METHOD Stop : BOOL
VAR_INPUT
END_VAR
tTimer_Enable(IN := FALSE);
tTimer_DropLid(IN := FALSE);
tTimer_Suction(IN := FALSE);
tTimer_TakeLid(IN := FALSE);
tTimer_Pick(IN := FALSE);
iCylinder_LidStopper.Extend();
iLidSuctionValve.Release();
iCupSuctionValve.Release();
END_METHOD

METHOD TakeLid : BOOL
VAR_INPUT
END_VAR
CASE nState_TakeLid OF
	0://init
		TakeLid := FALSE;
		tTimer_TakeLid(IN:= FALSE);
		tTimer_Pick(IN := FALSE);
		nState_TakeLid := 1;
	1://check LidEmpty
		IF isLidPick THEN
			IF nLine = 1 THEN
				F_SetError(51,nLine := 1);
			ELSIF nLine = 2 THEN
				F_SetError(52,nLine := 2);
			END_IF
		ELSE
			nState_TakeLid := 11;
		END_IF
	11:// call cylinder_suction. retract to take lid
		iCylinder_Suction.Retract();
		IF iCylinder_Suction.bIsRetract THEN
			tTimer_TakeLid(IN := FALSE);
			nState_TakeLid := 2;
		ELSE
			tTimer_TakeLid(IN := TRUE, PT := REAL_TO_TIME(timerCylinder_Suction)*1000);
			IF tTimer_TakeLid.Q THEN
				IF nLine = 1 THEN
					F_SetError(13,nLine := 1);
				ELSIF nLine = 2 THEN
					F_SetError(35,nLine := 2);
				END_IF
			END_IF
		END_IF
	2://call cylinder_Lidstop.retract to drop lid
		iCylinder_LidStopper.Retract();
		IF iCylinder_LidStopper.bIsRetract THEN
			tTimer_TakeLid(IN := FALSE);
			nState_TakeLid := 3;
		ELSE
			tTimer_TakeLid(IN := TRUE, PT := REAL_TO_TIME(timerCylinder_Stopper)*1000);
			IF tTimer_TakeLid.Q THEN
				IF nLine = 1 THEN
					F_SetError(11,nLine := 1);
				ELSIF nLine = 2 THEN
					F_SetError(33,nLine := 2);
				END_IF
			END_IF
		END_IF
	3:// Suck lid
		iCylinder_LidStopper.Retract();
		iLidSuctionValve.Suck();
		IF isLidPick THEN
			tTimer_TakeLid(IN := FALSE);
			nState_TakeLid := 33;
		ELSE
			tTimer_TakeLid(IN := TRUE, PT := REAL_TO_TIME(timerCheckLidSuck)*1000);
			IF tTimer_TakeLid.Q THEN
				IF nLine = 1 THEN
					F_SetError(49,nLine := 1);
					nState_TakeLid := 2;
				ELSIF nLine = 2 THEN
					F_SetError(50,nLine := 2);
					nState_TakeLid := 2;
				END_IF
			END_IF
		END_IF
	33:
		iLidSuctionValve.Suck();
		tTimer_Pick(IN := TRUE, PT:= T#0.5S);
		IF tTimer_Pick.Q THEN
			nState_TakeLid := 4;
		END_IF
	4://Block Lid Up
		iLidSuctionValve.Suck();
		tTimer_Pick(IN := FALSE);
		iCylinder_LidStopper.Extend();
		IF iCylinder_LidStopper.bIsExtend THEN
			tTimer_TakeLid(IN := FALSE);
			nState_TakeLid := 5;
		ELSE
			tTimer_TakeLid(IN := TRUE, PT := REAL_TO_TIME(timerCylinder_Stopper)*1000);
			IF tTimer_TakeLid.Q THEN
				IF nLine = 1 THEN
					F_SetError(12,nLine := 1);
				ELSIF nLine = 2 THEN
					F_SetError(34,nLine := 2);
				END_IF
			END_IF
		END_IF
	5://finish takelid
		TakeLid := TRUE;
		nState_TakeLid := 0;	
END_CASE
END_METHOD

END_FUNCTION_BLOCK

// ---- POUs/Components/Child Components/FB_SuctionCup.TcPOU
FUNCTION_BLOCK FB_SuctionCup IMPLEMENTS I_SuctionCup
VAR_INPUT
END_VAR
VAR_OUTPUT
END_VAR
VAR
	fPressure 		AT %I*	: REAL;
	bSuck			AT %Q*	: BOOL;
	bPressure		AT %I* 	: BOOL;
END_VAR

PROPERTY bIsSuck : BOOL
GET
bIsSuck := bPressure;
END_GET
END_PROPERTY

PROPERTY fThreshold : REAL
GET
fThreshold := 6;
END_GET
SET
END_SET
END_PROPERTY

METHOD Release : BOOL
VAR_INPUT
END_VAR
bSuck := FALSE;
END_METHOD

METHOD Suck : BOOL
VAR_INPUT
END_VAR
bSuck := TRUE;
END_METHOD

END_FUNCTION_BLOCK

// ---- POUs/Components/Sim Components/FB_SuctionCup_Sim.TcPOU
FUNCTION_BLOCK FB_SuctionCup_Sim IMPLEMENTS I_SuctionCup
VAR_INPUT
END_VAR
VAR_OUTPUT
END_VAR
VAR
	fPressure 			: REAL;// Value 0-100 %
	bSuck				: BOOL;
	// var sim
	tTimer				: TON;
	tDelay				: TIME := T#1000MS;// acceleration time of fPressure to value = 100
	nState				: INT := 0;
	bRelease			: BOOL := TRUE;
END_VAR

CASE nState OF
	0: //init release Suction
		IF bRelease THEN
			bSuck := FALSE;
			fPressure := 0;
		ELSE
			bSuck := TRUE;
			fPressure := 100;
		END_IF
		tTimer(IN := FALSE);
		nState := nState + 1;
	1:// check for signal
		tTimer(IN := FALSE);
		IF bSuck AND (fPressure = 0) THEN
			nState := 10;
		END_IF
		IF NOT bSuck AND (fPressure = 100) THEN
			nState := 20;
		END_IF
	10: //Suck 
		tTimer(IN := TRUE,PT := tDelay);
		fPressure := TIME_TO_REAL(tTimer.ET)*(100/TIME_TO_REAL(tDelay));
		IF (fPressure = 100) THEN
			nState := 1;
		END_IF
	20:// release
		tTimer(IN := TRUE,PT := tDelay);
		fPressure := 100 - (TIME_TO_REAL(tTimer.ET)*(100/TIME_TO_REAL(tDelay)));
		IF (fPressure = 0) THEN
			nState := 1;
		END_IF
END_CASE

PROPERTY bIsSuck : BOOL
GET
IF fPressure > fThreshold THEN
	bIsSuck := TRUE;
ELSE 
	bIsSuck := FALSE;
END_IF
END_GET
END_PROPERTY

PROPERTY fThreshold : REAL
GET
fThreshold := 50;
END_GET
SET
END_SET
END_PROPERTY

METHOD Release : BOOL
VAR_INPUT
END_VAR
bSuck := FALSE;
END_METHOD

METHOD Suck : BOOL
VAR_INPUT
END_VAR
bSuck := TRUE;
END_METHOD

END_FUNCTION_BLOCK

// ---- POUs/Modules/FB_LidCloseModule.TcPOU
FUNCTION_BLOCK FB_LidCloseModule
VAR_INPUT
	nLine							: INT;
	timer_Check_Cylinder_extend		: REAL;
	timer_Check_Cylinder_retract	: REAL;
	timer_CloseLid					: REAL;
END_VAR
VAR_OUTPUT
END_VAR
VAR
	// ===== CHILD COMPONENTS ======
	fbCylinder_LidClose 		: FB_Cylinder;
	// ===== SIM COMPONENTS ======
	fbCylinder_LidClose_Sim		: FB_Cylinder_Sim;
	// ===== INTERFACES ======
	iCylinder					: I_Cylinder;
	// ===== Var method enable
	nState_Enable				: INT;
	tTimer_Enable				: TON;
	// ===== Var method CloseLid
	nState_Close				: INT;
	tTimer_Close				: TON;
	i							: INT := 1; //number of repetitions
END_VAR

IF bSimMode THEN
	iCylinder := fbCylinder_LidClose_Sim;
	fbCylinder_LidClose_Sim();
ELSE
	iCylinder := fbCylinder_LidClose;
	fbCylinder_LidClose(id := 1);
END_IF

METHOD CloseLid : BOOL
VAR_INPUT
END_VAR
CASE nState_Close OF
	0:
		CloseLid := FALSE;
		tTimer_Close(IN := FALSE);
		nState_Close := 1;
	1: //set init i
		i := 1;
		nState_Close := 2;
	2: // cylinder extend and check sensor
		iCylinder.Extend();
		IF iCylinder.bIsExtend THEN
			tTimer_Close(IN := FALSE);
			nState_Close := 3;
		ELSE
			tTimer_Close(IN := TRUE,PT := REAL_TO_TIME(timer_Check_Cylinder_extend)*1000);
			IF tTimer_Close.Q THEN
				i := i + 1;
				nState_Close := 3;
			END_IF
		END_IF
	3: //cylinder retract
		iCylinder.Retract();
		IF iCylinder.bIsRetract THEN
			tTimer_Close(IN := FALSE);
			nState_Close := 4;//return extend
		ELSE
			tTimer_Close(IN := TRUE,PT := REAL_TO_TIME(timer_Check_Cylinder_retract)*1000);
			IF tTimer_Close.Q THEN
				IF nLine = 1 THEN
					F_SetError(15,nLine := 1);
				ELSIF nLine = 2 THEN
					F_SetError(37,nLine := 2);
				END_IF
			END_IF
		END_IF
	4:// cylinder extend and check sensor
		iCylinder.Extend();
		IF iCylinder.bIsExtend THEN
			tTimer_Close(IN := FALSE);
			nState_Close := 5;
		ELSE
			tTimer_Close(IN := TRUE,PT := REAL_TO_TIME(timer_Check_Cylinder_extend)*1000);
			IF tTimer_Close.Q THEN
				i := i + 1;
				nState_Close := 5;
			END_IF
		END_IF
	5:// cylinder retract -> end
		iCylinder.Retract();
		IF iCylinder.bIsRetract THEN
			tTimer_Close(IN := FALSE);
			nState_Close := 6;//end
		ELSE
			tTimer_Close(IN := TRUE,PT := REAL_TO_TIME(timer_Check_Cylinder_retract)*1000);
			IF tTimer_Close.Q THEN
				IF nLine = 1 THEN
					F_SetError(15,nLine := 1);
				ELSIF nLine = 2 THEN
					F_SetError(37,nLine := 2);
				END_IF
			END_IF
		END_IF
	6://check warning
		IF (i = 3) THEN
			IF nLine = 1 THEN
				F_SetWarning(107,nLine := 1);
			ELSIF nLine = 2 THEN 
				F_SetWarning(114,nLine := 2);
			END_IF
			
			nState_Close := 7; //end
		ELSE
			nState_Close := 7; //end
		END_IF
	7: //Finish
		CloseLid := TRUE;
		nState_Close := 0;
END_CASE
END_METHOD

METHOD Enable : BOOL
VAR_INPUT
END_VAR
CASE nState_Enable OF
	0:
		Enable 			:= FALSE;
		tTimer_Enable(IN := FALSE);
		nState_Enable 	:= 1;
	1: // cylinder retract and check
		iCylinder.Retract();
		IF iCylinder.bIsRetract THEN
			tTimer_Enable(IN := FALSE);
			nState_Enable 	:= 2;
		ELSE
			tTimer_Enable(IN := TRUE, PT := REAL_TO_TIME(timer_Check_Cylinder_retract)*1000);
			IF tTimer_Enable.Q THEN
				IF nLine = 1 THEN
					F_SetError(15,nLine := 1);
				ELSIF nLine = 2 THEN
					F_SetError(33,nLine := 2);
				END_IF
			END_IF
		END_IF
	2:
		tTimer_Enable(IN := FALSE);
		Enable := TRUE;
	99://Error
END_CASE
END_METHOD

METHOD Init : BOOL
VAR_INPUT
END_VAR
nState_Close := 0;
i 			 := 1;
END_METHOD

METHOD Manual : BOOL
VAR_INPUT
	bCylinder_CloseLid_Extend	: BOOL;
	bCylinder_CloseLid_Retract	: BOOL;
END_VAR
IF bCylinder_CloseLid_Extend THEN
	iCylinder.Extend();
	IF iCylinder.bIsExtend THEN
		tTimer_Close(IN := FALSE);
	ELSE
		tTimer_Close(IN := TRUE,PT := REAL_TO_TIME(timer_Check_Cylinder_retract)*1000);
		IF tTimer_Close.Q THEN
			IF nLine = 1 THEN
				F_SetError(16,nLine := 1);
			ELSIF nLine = 2 THEN
				F_SetError(38,nLine := 2);
			END_IF
		END_IF
	END_IF
ELSIF bCylinder_CloseLid_Retract THEN
	iCylinder.Retract();
	IF iCylinder.bIsRetract THEN
		tTimer_Close(IN := FALSE);
	ELSE
		tTimer_Close(IN := TRUE,PT := REAL_TO_TIME(timer_Check_Cylinder_retract)*1000);
		IF tTimer_Close.Q THEN
			IF nLine = 1 THEN
				F_SetError(15,nLine := 1);
			ELSIF nLine = 2 THEN
				F_SetError(37,nLine := 2);
			END_IF
		END_IF
	END_IF
END_IF
END_METHOD

METHOD Reset : BOOL
VAR_INPUT
END_VAR
tTimer_Enable(IN := FALSE);							
tTimer_Close(IN := FALSE);
iCylinder.Retract();
END_METHOD

METHOD Stop : BOOL
VAR_INPUT
END_VAR
tTimer_Enable(IN := FALSE);						
tTimer_Close(IN := FALSE);
END_METHOD

END_FUNCTION_BLOCK

// ---- POUs/Modules/FB_Transfer.TcPOU
FUNCTION_BLOCK FB_Transfer
VAR_INPUT
	nLine					: INT;
	fTimer_Comb				: REAL;
	fTimer_Clip				: REAL;
	fTimer_Move_Comb		: REAL;
END_VAR
VAR_OUTPUT
	nDoneTransfer			: INT;
	bDoneTransfer			: BOOL;
END_VAR
VAR
	fbCylinder_Comb			: FB_Cylinder;
	fbCylinder_Clip			: FB_Cylinder;
	fbCylinder_Move_Comb	: FB_Cylinder;
	// ===== SIM COMPONENTS ==============
	fbCylinderSim_Comb		: FB_Cylinder_Sim;
	fbCylinderSim_Clip		: FB_Cylinder_Sim;
	fbCylinderSim_Move_Comb	: FB_Cylinder_Sim;
	// ===== INTERFACES ==================
	iCylinder_Comb			: I_Cylinder;
	iCylinder_Clip			: I_Cylinder;
	iCylinder_Move_Comb		: I_Cylinder;
	//====== VAR MOTHOD ==================
	nState					: INT;
	nStateEnable			: INT;
	nState_Reset			: INT;
	tTimer_Reset			: TON;
	fbTimer_Comb			: TON;
	fbTimer_Clip			: TON;
	fbTimer_Move_Comb		: TON;
	//======== VAR HMI Transfer Setting ====
END_VAR

IF bSimMode THEN
	iCylinder_Clip 	:= fbCylinderSim_Clip;
	fbCylinderSim_Clip();
	iCylinder_Comb	:= fbCylinderSim_Comb;
	fbCylinderSim_Comb();
	iCylinder_Move_Comb	:= fbCylinderSim_Move_Comb;
	fbCylinderSim_Move_Comb();
ELSE
	iCylinder_Clip 	:= fbCylinder_Clip;
	fbCylinder_Clip(id := 1);
	iCylinder_Comb	:= fbCylinder_Comb;
	fbCylinder_Comb(id := 1);
	iCylinder_Move_Comb	:= fbCylinder_Move_Comb;
	fbCylinder_Move_Comb(id := 1);
END_IF

METHOD Auto : BOOL
VAR_INPUT
END_VAR
fbTimer_Clip(PT := REAL_TO_TIME(fTimer_Clip)*1000);
fbTimer_Comb(PT := REAL_TO_TIME(fTimer_Comb)*1000);
fbTimer_Move_Comb(PT := REAL_TO_TIME(fTimer_Move_Comb)*1000);
CASE nState OF 
	0: // init value
		Auto		:= FALSE;
		fbTimer_Move_Comb(IN := FALSE);
		fbTimer_Clip(IN	:= FALSE);
		fbTimer_Comb(IN	:= FALSE);
		nState		:= 1;
	1: // Cylinder Clip and Comb Extend hold cup
		bDoneTransfer 	:= FALSE;
		iCylinder_Clip.Extend();
		iCylinder_Comb.Extend();
		fbTimer_Clip(IN	:= TRUE);
		fbTimer_Comb(IN	:= TRUE);
		IF iCylinder_Clip.bIsExtend AND iCylinder_Comb.bIsExtend THEN
			nState	:= 2;
		ELSIF fbTimer_Comb.Q AND NOT fbTimer_Clip.Q THEN
			IF nLine = 1 THEN
				F_SetError(18,nLine := 1);
			ELSIF nLine = 2 THEN
				F_SetError(40,nLine := 2);
			END_IF
		ELSIF fbTimer_Clip.Q AND NOT fbTimer_Comb.Q THEN
			IF nLine = 1 THEN
				F_SetError(20,nLine := 1);
			ELSIF nLine = 2 THEN
				F_SetError(42,nLine := 2);
			END_IF
		ELSIF iCylinder_Clip.bIsExtend AND fbTimer_Comb.Q THEN
			IF nLine = 1 THEN
				F_SetError(18,nLine := 1);
			ELSIF nLine = 2 THEN
				F_SetError(40,nLine := 2);
			END_IF
		ELSIF iCylinder_Comb.bIsExtend AND fbTimer_Clip.Q THEN
			IF nLine = 1 THEN
				F_SetError(20,nLine := 1);
			ELSIF nLine = 2 THEN
				F_SetError(42,nLine := 2);
			END_IF
		ELSIF fbTimer_Comb.Q AND fbTimer_Clip.Q THEN
			IF nLine = 1 THEN
				F_SetError(18,nLine := 1);
			ELSIF nLine = 2 THEN
				F_SetError(40,nLine := 2);
			END_IF
		END_IF
	2: // Cylinder_Move_Comb Extend move cup
		fbTimer_Clip(IN	:= FALSE);
		fbTimer_Comb(IN	:= FALSE);
		fbTimer_Move_Comb(IN := TRUE);
		iCylinder_Move_Comb.Extend();
		IF iCylinder_Move_Comb.bIsExtend THEN
			nState	:= 3;
		ELSIF fbTimer_Move_Comb.Q THEN
			IF nLine = 1 THEN
				F_SetError(22,nLine := 1);
			ELSIF nLine = 2 THEN
				F_SetError(44,nLine := 2);
			END_IF
		END_IF
	3: // retract clip and comb
		fbTimer_Comb(IN := TRUE);
		fbTimer_Move_Comb(IN := FALSE);
		iCylinder_Comb.Retract();
		IF iCylinder_Comb.bIsRetract THEN
			nState	:= 33;
		ELSIF fbTimer_Comb.Q THEN
			IF nLine = 1 THEN
				F_SetError(17,nLine := 1);
			ELSIF nLine = 2 THEN
				F_SetError(39,nLine := 2);
			END_IF
		END_IF
	33:
		fbTimer_Clip(IN := TRUE);
		fbTimer_Comb(IN := FALSE);
		iCylinder_Clip.Retract();
		IF iCylinder_Clip.bIsRetract THEN
			nDoneTransfer	:= nDoneTransfer + 1;
			bDoneTransfer 	:= TRUE;
			IF nLine = 1 THEN 
				bToDropcup1			:= TRUE;
			ELSIF nLine = 2 THEN
				bToDropcup2			:= TRUE;
			END_IF
			IF nDoneTransfer > 8 THEN
				nDoneTransfer := 8;
			END_IF
			nState	:= 4;
		ELSIF fbTimer_Clip.Q THEN
			IF nLine = 1 THEN
				F_SetError(19,nLine := 1);
			ELSIF nLine = 2 THEN
				F_SetError(41,nLine := 2);
			END_IF
		END_IF
	4://Move_Comb Retract
		fbTimer_Clip(IN := FALSE);
		fbTimer_Move_Comb(IN := TRUE);
		iCylinder_Move_Comb.Retract();
		IF iCylinder_Move_Comb.bIsRetract THEN
			nState	:= 5;
		ELSIF fbTimer_Move_Comb.Q THEN
			IF nLine = 1 THEN
				F_SetError(21,nLine := 1);
			ELSIF nLine = 2 THEN
				F_SetError(43,nLine := 2);
			END_IF
		END_IF
	5:// Complete
		fbTimer_Move_Comb(IN := FALSE);
		Auto		:= TRUE;
		nState		:= 0;	
END_CASE
END_METHOD

METHOD Enable : BOOL
VAR_INPUT
END_VAR
fbTimer_Clip(PT := REAL_TO_TIME(fTimer_Clip)*1000);
fbTimer_Comb(PT := REAL_TO_TIME(fTimer_Comb)*1000);
fbTimer_Move_Comb(PT := REAL_TO_TIME(fTimer_Move_Comb)*1000);
CASE nStateEnable OF
	0:// init 
		Enable					:= FALSE;
		fbTimer_Clip(IN	:= FALSE);
		fbTimer_Comb(IN	:= FALSE);
		fbTimer_Move_Comb(IN := FALSE);
		nStateEnable			:= 1;
	1:// Retract Comb and Clip
		iCylinder_Clip.Retract();
		iCylinder_Comb.Retract();
		fbTimer_Clip(IN	:= TRUE);
		fbTimer_Comb(IN	:= TRUE);
		IF iCylinder_Clip.bIsRetract AND iCylinder_Comb.bIsRetract THEN
			nStateEnable		:= 2;
		ELSIF fbTimer_Clip.Q AND NOT fbTimer_Comb.Q THEN
			nStateEnable		:= 10;
		ELSIF fbTimer_Comb.Q AND NOT fbTimer_Clip.Q THEN
			nStateEnable		:= 11;
		END_IF	
	2:// Retract MoveComb
		fbTimer_Clip(IN	:= FALSE);
		fbTimer_Comb(IN	:= FALSE);
		iCylinder_Move_Comb.Retract();
		fbTimer_Move_Comb.IN	:= TRUE;
		IF iCylinder_Move_Comb.bIsRetract THEN
			nStateEnable		:= 3;
		ELSIF fbTimer_Move_Comb.Q THEN
			nState				:= 12;
		END_IF
	3:// Enable
		fbTimer_Move_Comb(IN := FALSE);
		Enable					:= TRUE;
	10:// Error Cylinder Clip
		IF nLine = 1 THEN
			F_SetError(17,nLine := 1);
			nState	:= 99;
		ELSIF nLine = 2 THEN
			F_SetError(35,nLine := 2);
			nState	:= 99;
		END_IF
	11:// Error Cylinder Comb
		IF nLine = 1 THEN
			F_SetError(16,nLine := 1);
			nState	:= 99;
		ELSIF nLine = 2 THEN
			F_SetError(34,nLine := 2);
			nState	:= 99;
		END_IF
	12:// Error Cylinder MoveComb
		IF nLine = 1 THEN
			F_SetError(18,nLine := 1);
			nState	:= 99;
		ELSIF nLine = 2 THEN
			F_SetError(36,nLine := 2);
			nState	:= 99;
		END_IF
	99:// Error
END_CASE
END_METHOD

METHOD Init : BOOL
VAR_INPUT
END_VAR
nState		 := 0;
nStateEnable := 0;
bDoneTransfer := FALSE;
nDoneTransfer := 0;
END_METHOD

METHOD Manual : BOOL
VAR_INPUT
	bCylinder_Comb_Extend			: BOOL;
	bCylinder_Comb_Retract			: BOOL;
	bCylinder_Clip_Extend			: BOOL;
	bCylinder_Clip_Retract			: BOOL;
	bCylinder_Move_Comb_Extend		: BOOL;
	bCylinder_Move_Comb_Retract		: BOOL;
END_VAR
IF bCylinder_Comb_Extend THEN
	iCylinder_Comb.Extend();
	IF iCylinder_Comb.bIsExtend THEN
		fbTimer_Comb(IN := FALSE);
	ELSE
		fbTimer_Comb(PT := REAL_TO_TIME(fTimer_Comb)*1000);
			IF fbTimer_Comb.Q THEN
				IF nLine = 1 THEN
					F_SetError(18,nLine := 1);
				ELSIF nLine = 2 THEN
					F_SetError(40,nLine := 2);
				END_IF
			END_IF
	END_IF
END_IF

IF bCylinder_Comb_Retract THEN
	iCylinder_Comb.Retract();
	IF iCylinder_Comb.bIsRetract THEN
		fbTimer_Comb(IN := FALSE);
	ELSE
		fbTimer_Comb(PT := REAL_TO_TIME(fTimer_Comb)*1000);
			IF fbTimer_Comb.Q THEN
				IF nLine = 1 THEN
					F_SetError(17,nLine := 1);
				ELSIF nLine = 2 THEN
					F_SetError(39,nLine := 2);
				END_IF
			END_IF
	END_IF
END_IF

IF bCylinder_Clip_Extend THEN
	iCylinder_Clip.Extend();
	IF iCylinder_Clip.bIsExtend THEN
		fbTimer_Clip(IN := FALSE);
	ELSE
		fbTimer_Clip(PT := REAL_TO_TIME(fTimer_Clip)*1000);
			IF fbTimer_Clip.Q THEN
				IF nLine = 1 THEN
					F_SetError(20,nLine := 1);
				ELSIF nLine = 2 THEN
					F_SetError(42,nLine := 2);
				END_IF
			END_IF
	END_IF
END_IF


IF bCylinder_Clip_Retract THEN
	iCylinder_Clip.Retract();	
	IF iCylinder_Clip.bIsRetract THEN
		fbTimer_Clip(IN := FALSE);
	ELSE
		fbTimer_Clip(PT := REAL_TO_TIME(fTimer_Clip)*1000);
			IF fbTimer_Clip.Q THEN
				IF nLine = 1 THEN
					F_SetError(19,nLine := 1);
				ELSIF nLine = 2 THEN
					F_SetError(41,nLine := 2);
				END_IF
			END_IF
	END_IF
END_IF

IF bCylinder_Move_Comb_Extend THEN
	iCylinder_Move_Comb.Extend();
	IF iCylinder_Move_Comb.bIsExtend THEN
		fbTimer_Move_Comb(IN := FALSE);
	ELSE
		fbTimer_Move_Comb(PT := REAL_TO_TIME(fTimer_Move_Comb)*1000);
			IF fbTimer_Move_Comb.Q THEN
				IF nLine = 1 THEN
					F_SetError(22,nLine := 1);
				ELSIF nLine = 2 THEN
					F_SetError(44,nLine := 2);
				END_IF
			END_IF
	END_IF
END_IF

IF bCylinder_Move_Comb_Retract THEN
	iCylinder_Move_Comb.Retract();
	IF iCylinder_Move_Comb.bIsRetract THEN
		fbTimer_Move_Comb(IN := FALSE);
	ELSE
		fbTimer_Move_Comb(PT := REAL_TO_TIME(fTimer_Move_Comb)*1000);
			IF fbTimer_Move_Comb.Q THEN
				IF nLine = 1 THEN
					F_SetError(21,nLine := 1);
				ELSIF nLine = 2 THEN
					F_SetError(43,nLine := 2);
				END_IF
			END_IF
	END_IF
END_IF
END_METHOD

METHOD Reset : BOOL
VAR_INPUT
END_VAR
iCylinder_Clip.Retract();
fbTimer_Clip(IN	:= FALSE);
fbTimer_Comb(IN	:= FALSE);
fbTimer_Move_Comb(IN := FALSE);

CASE nState_Reset OF
	0:
		iCylinder_Comb.Retract();
		tTimer_Reset(IN := TRUE, PT := T#300MS);
		IF tTimer_Reset.Q OR iCylinder_Comb.bIsRetract THEN
			nState_Reset := 1;
		END_IF
	1:
		iCylinder_Move_Comb.Retract();
		nState_Reset := 0;
END_CASE
END_METHOD

METHOD Stop : BOOL
VAR_INPUT
END_VAR
fbTimer_Clip(IN	:= FALSE);
fbTimer_Comb(IN	:= FALSE);
fbTimer_Move_Comb(IN := FALSE);
END_METHOD

END_FUNCTION_BLOCK

// ---- POUs/Machines/PR_Line02.TcPOU
PROGRAM PR_Line02
VAR PERSISTENT
//----------------VAR SETTING--------------------
	timerCheckCylinder_Up			: REAL;//CupSupply
	timerCheckCylinder_Dw			: REAL;
	timerCheckEmpty					: REAL;
	timerCheckStuck					: REAL;
	timerCylinder_Up_extend 		: REAL;
	timerCylinder_Suction_Cup_extend: REAL;
	timerCylinder_Suction_Cup		: REAL;
	timerCylinder_Suction_Val		: REAL;
	timerCylinder_Suction_pick		: REAL;
	fSpeed_motor_mixer				: REAL;//FoodMixer
	fTimer_Reverse					: REAL;
	fFast_Speed						: REAL;//FoodWeight
	fSlow_Speed_1					: REAL;
	fSlow_Speed_2					: REAL;
	fDerisedWeight_Food				: REAL;
	fChangeMode_Food_1				: REAL;
	fChangeMode_Food_2				: REAL;
	fMaxWeight_Food					: REAL;
	fPerStop_Food					: REAL;
	fTimer_Food						: REAL;
	fTimer_Alarm_Food				: REAL;
	fTimer_Check_Food				: REAL;
	fDelta_Food						: REAL;
	fTimer_rever_food				: REAL;
	fTimer_Error_Food				: REAL;
	fFast_Speed_vibrating_funnel	: REAL;//WormWeight
	fSlow_Speed_vibrating_funnel_1	: REAL;
	fSlow_Speed_vibrating_funnel_2	: REAL;
	fDerisedWeight_Worm				: REAL;
	fChangeMode_Worm_1				: REAL;
	fChangeMode_Worm_2				: REAL;
	fMaxWeight_Worm					: REAL;
	fPerStop_Worm					: REAL;
	fTimer_Worm						: REAL;
	fTimer_Alarm_Worm				: REAL;
	fTimer_Check_Worm				: REAL;
	fTimer_Check_Cylinder			: REAL;
	fDelta_Worm						: REAL;
	fTimer_Error_Worm				: REAL;
	timerCylinder_Suction			: REAL;//LidSupply
	timerCheckLidRelease			: REAL;
	timerLidBlow					: REAL;
	timerCheckLidEmpty				: REAL;
	timerCheckLidSuck				: REAL;
	timerCylinder_Stopper			: REAL;
	timer_Check_Cylinder_extend		: REAL;//LidClose
	timer_Check_Cylinder_retract	: REAL;
	timer_CloseLid					: REAL;
	fTimer_Comb						: REAL;//Transfer
	fTimer_Clip						: REAL;
	fTimer_Move_Comb				: REAL;
//-----------------VAR HMI-------------------
	fProductLog						: ARRAY [1..2] OF ARRAY  [1..5] OF REAL;
END_VAR

VAR
	bStatus_Food					: BOOL;
	bStatus_Worm					: BOOL;
//----------------VAR MANUAL---------------------
	bCylinder_up_extend 			: BOOL;//CupSupply
	bCylinder_up_retract 			: BOOL;
	bCylinder_dw_extend 			: BOOL;
	bCylinder_dw_retract 			: BOOL;
	bCylinder_Suction_cup_extend	: BOOL;
	bCylinder_Suction_cup_retract	: BOOL;
	bUp_Motor_Mixer					: BOOL;//FoodMixer
	bDown_Motor_Mixer				: BOOL;
	bMotor_mixer_Manual				: BOOL;
	bMotor_mixer_reverse			: BOOL;
	bUp_Food_Motor					: BOOL;//FoodWeight
	bDown_Food_Motor				: BOOL;
	bZero_Loadcell_Food				: BOOL;
	bMotor_Food						: BOOL;
	bMotor_Food_reverse				: BOOL;
	bUp_vibrating_funnel			: BOOL;//WormWeight
	bDown_vibrating_funnel			: BOOL;
	bZero_Loadcell_Worm				: BOOL;
	bCylinder_Block_Worm_Extend		: BOOL;
	bCylinder_Block_Worm_Retract	: BOOL;
	bMotor_vibrating_funnel			: BOOL;	
	bCylinder_LidStopper_extend 	: BOOL;//LidSupply
	bCylinder_LidStopper_retract 	: BOOL;
	bCylinder_Suction_extend		: BOOL;
	bCylinder_Suction_retract		: BOOL;
	bLidSuctionValve				: BOOL;
	bCupSuctionValve				: BOOL;
	bBlowValve						: BOOL;
	bCylinder_CloseLid_Extend		: BOOL;//LidClose
	bCylinder_CloseLid_Retract		: BOOL;
	bCylinder_Comb_Extend			: BOOL;//Transfer
	bCylinder_Comb_Retract			: BOOL;
	bCylinder_Clip_Extend			: BOOL;
	bCylinder_Clip_Retract			: BOOL;
	bCylinder_Move_Comb_Extend		: BOOL;
	bCylinder_Move_Comb_Retract		: BOOL;
//------------------fbmodule----------------
	fb_CupSupply	: FB_CupSupplyModule;
	fb_FoodMixer	: FB_FoodMixerModule;
	fb_FoodWeight	: FB_FoodWeightModule;
	fb_WormWeight	: FB_WormWeightModule;
	fb_LidSupply	: FB_LidSupplyModule;
	fb_LidClose		: FB_LidCloseModule;
	fb_Transfer		: FB_Transfer;
//---------------- VAR Method ---------------
	nState				: INT;
	nState_Dropcup		: INT;
	nState_Transfer		: INT;
	nState_FoodWeight	: INT;
	nState_WormWeight	: INT;
	nState_LidClose		: INT;
	nState_LidSupply	: INT;
	nDoneTransfer		: INT;
	nDoneTransferStop	: INT;
	tmp					: INT;
	bDoneTakeLid		: BOOL;
	bDoneTransfer		: BOOL;
	bDoneCupSupply		: BOOL;
	bDoneFoodWeight		: BOOL;
	bDoneWormWeight		: BOOL;
	bDoneLidSupply		: BOOL;
	bDoneLidClose		: BOOL;
	bEnable				: BOOL;
	bFinishCupSupply	: BOOL;
	bFinishFoodWeight	: BOOL;
	bFinishWormWeight	: BOOL;
	bFinishLidSupply	: BOOL;
	bFinishLidClose		: BOOL;
	bFinishTransfer		: BOOL;
	//-------VAR--------------
	nStateConveyor		: INT;
	fbtimertransfer		: TON;
	fbTimer				: TON;
	nStateStop			: INT;
	fbtimerStop			: ton;
	fbTimerCycle		: ton;
	timeCycle			: REAL :=1;
	fproduct			: INT;
	nstateCycle			: INT;
	bDone				: R_TRIG;
	fbDelay				: TON;
	bStatus_Food_order	: ARRAY [1..3] OF BOOL;
	bStatus_Worm_order	: ARRAY [1..3] OF BOOL;
	bStatus_Lid_order	: ARRAY [1..3] OF BOOL;
	i1,i2,i3			: INT := 0;
	xathucan			: BOOL;
	xasau				: BOOL;
	daothucan			: BOOL;
	nstatetest1			: INT;
	nstatetest2			: INT;
	nstatetest3			: INT;
	bxa					: BOOL;
	bCheck				: BOOL;
	bypassFood			: BOOL;
	bypassWorm			: BOOL;
	bypassLid			: BOOL;
END_VAR

fb_CupSupply(
	nLine:= 2 , 
	timerCheckCylinder_Up:= timerCheckCylinder_Up, 
	timerCheckCylinder_Dw:= timerCheckCylinder_Dw, 
	timerCheckEmpty:= timerCheckEmpty, 
	timerCheckStuck:= timerCheckStuck,
	timerCylinder_Up_extend := timerCylinder_Up_extend,
	timerCylinder_Suction:= timerCylinder_Suction_Cup,
	timerCylinder_Suction_extend:= timerCylinder_Suction_Cup_extend,
	ttimerCylinder_val:=timerCylinder_Suction_Val,
	timerCylinder_Suction_pick:=timerCylinder_Suction_pick);

fb_FoodMixer(
	nLine:= 2,
	UnitID:= 1, 
	fSpeed_motor_mixer:= fSpeed_motor_mixer,
	fTimer_Reverse:= fTimer_Reverse);
		
fb_FoodWeight(
	nLine:= 2, 
	UnitID:= 6, 
	fFast_Speed:= fFast_Speed, 
	fSlow_Speed_1:= fSlow_Speed_1, 
	fSlow_Speed_2:= fSlow_Speed_2, 
	fDerisedWeight_Food:= fDerisedWeight_Food, 
	fChangeMode_Food_1:= fChangeMode_Food_1, 
	fChangeMode_Food_2:= fChangeMode_Food_2, 
	fMaxWeight_Food:= fMaxWeight_Food, 
	fPerStop_Food:= fPerStop_Food, 
	fTimer_Food:= fTimer_Food, 
	fTimer_Alarm_Food:= fTimer_Alarm_Food, 
	fTimer_Check_Food:= fTimer_Check_Food, 
	fDelta_Food:= fDelta_Food,
	fTimer_Reverse := fTimer_rever_food,
	fTimer_Error_Food := fTimer_Error_Food, 
	fProductLogF=> fProductLog[1],
	bStatus_Food=> bStatus_Food,
	Time_start=>Time_Start_Food_line2,
	Time_Stop=>Time_Stop_Food_line2,
	status=>bStatus_Food_line2,
	fweight_iot =>fWeight_Food_line2);

fb_LidClose(
	nLine:= 2, 
	timer_Check_Cylinder_extend:= timer_Check_Cylinder_extend, 
	timer_Check_Cylinder_retract:= timer_Check_Cylinder_retract, 
	timer_CloseLid:= timer_CloseLid);
	
fb_LidSupply(
	nLine:= 2, 
	timerCylinder_Suction:= timerCylinder_Suction, 
	timerCheckLidRelease:= timerCheckLidRelease, 
	timerLidBlow:= timerLidBlow, 
	timerCheckLidEmpty:= timerCheckLidEmpty, 
	timerCheckLidSuck:= timerCheckLidSuck, 
	timerCylinder_Stopper:= timerCylinder_Stopper);

fb_Transfer(
	nLine:= 2, 
	fTimer_Comb:= fTimer_Comb, 
	fTimer_Clip:= fTimer_Clip, 
	fTimer_Move_Comb:= fTimer_Move_Comb, 
	nDoneTransfer=> nDoneTransfer,
	bDoneTransfer=> bDoneTransfer);

fb_WormWeight(
	nLine:= 2, 
	UnitID:= 2, 
	fFast_Speed_vibrating_funnel:= fFast_Speed_vibrating_funnel, 
	fSlow_Speed_vibrating_funnel_1:= fSlow_Speed_vibrating_funnel_1, 
	fSlow_Speed_vibrating_funnel_2:= fSlow_Speed_vibrating_funnel_2, 
	fDerisedWeight_Worm:= fDerisedWeight_Worm, 
	fChangeMode_Worm_1:= fChangeMode_Worm_1, 
	fChangeMode_Worm_2:= fChangeMode_Worm_2, 
	fMaxWeight_Worm:= fMaxWeight_Worm, 
	fPerStop_Worm:= fPerStop_Worm, 
	fTimer_Worm:= fTimer_Worm, 
	fTimer_Alarm_Worm:= fTimer_Alarm_Worm, 
	fTimer_Check_Worm:= fTimer_Check_Worm, 
	fTimer_Check_Cylinder:= fTimer_Check_Cylinder, 
	fDelta_Worm:= fDelta_Worm, 
	fTimer_Error_Worm := fTimer_Error_Worm,
	fProductLog=> fProductLog[2],
	bStatus_Worm=>bStatus_Worm,
	Time_start=>Time_Start_Worm_line2,
	Time_Stop=>Time_Stop_Worm_line2,
	status=>bStatus_Worm_line2,
	fweight_iot =>fWeight_Worm_line2);

IF bClear2 THEN
	nResult_false2 := 0;
	nResult_true2 := 0;
	nCount2 := 0;
	bClear2 := FALSE;
END_IF


fDerisedWeight_Food_line2	:= fDerisedWeight_Food;
fDerisedWeight_Worm_line2	:= fDerisedWeight_Worm;
fActDelta_Food_line2		:= fb_FoodWeight.fActDelta_Food;
fActDelta_Worm_line2		:= fb_WormWeight.fActDelta_Worm;
fDelta_Food_line2			:= fb_FoodWeight.fDelta_Food;
fDelta_Worm_line2			:= fb_WormWeight.fDelta_Worm;

IF getuser = 'Operator' THEN
	bypassFood := FALSE;
	bypassWorm := FALSE;
END_IF

ACTION Auto:
CASE nState OF
	0:// int
		bStatus_Food_order[1] := FALSE;
		bStatus_Worm_order[1] := FALSE;
		bStatus_Lid_order[1]  := FALSE;
		nDoneTransferStop	  := 0;
		fb_FoodWeight.SetZero();
		fb_WormWeight.SetZero();
		fb_Transfer.Init();
		i1 		:= 0;
		i2 		:= 0;
		i3 		:= 0;
		bfinish2:= TRUE;
		nState 	:= 1;
		
	1: // Start
		nState_FoodWeight := 0;
		nState_WormWeight := 0;
		nState_LidSupply := 0;
		nState_LidClose := 0;
		fb_FoodWeight.SetZero();
		fb_WormWeight.SetZero();
		bDoneCupSupply 		:= FALSE;
		bDoneFoodWeight 	:= FALSE;
		bDoneWormWeight 	:= FALSE;
		bDoneLidSupply 		:= FALSE;
		bDoneLidClose 		:= FALSE;
		bResetAuto2			:= FALSE;
		nState := 11;
	11:
		bStop2 := FALSE;
		bShift_is_over2 := FALSE;
		bStatusStart2 := FALSE;
		fb_FoodMixer.Stop();
		nStatus2	:= 'STOP';
		nState_Dropcup := 0;
		nState_Transfer := 0;
		bResetAuto2			:= FALSE;
		bFinishCupSupply 	:= FALSE;
		bFinishFoodWeight 	:= FALSE;
		bFinishWormWeight	:= FALSE;
		bFinishLidSupply	:= FALSE;
		bFinishLidClose		:= FALSE;
		bFinishTransfer		:= FALSE;
		bfinish2 := TRUE;
		nState := 22;
	22:
		IF bStart2 THEN
			bfinish2		:= FALSE;
			bStatusStart2	:= TRUE;
			bToDropcup2 	:= FALSE;
			bResetAuto2		:= TRUE;
			status			:= 'RUN';
			nState := 2;
		END_IF
			
	2: // start mode auto
		nStatus2	:= 'RUN';
		bResetAuto2		:= TRUE;
		bStart2		:= FALSE;
		bfinish2		:= FALSE;
		IF bypassfood THEN
			fb_FoodMixer.Stop();
		ELSE
			fb_FoodMixer.Auto();
		END_IF
		fb_CupSupply.CheckCup();
		fb_LidSupply.CheckLid();
		bDone(CLK := bDoneTransfer);
		CASE nstateCycle OF 
			0:
				fbTimerCycle(IN := TRUE, PT := T#100S);
				IF bDone.Q THEN
					nstateCycle := 1;
				END_IF
			1:
				timeCycle := TIME_TO_REAL(fbTimerCycle.ET)/1000;
				nstateCycle := 2;
			2: 
				fproduct := REAL_TO_INT(3600/(timeCycle+0.001));
				fbTimerCycle(IN := FALSE);
				nstateCycle := 0;
		END_CASE
		CASE nState_Dropcup OF
			0:// waiting for transfer
				fbDelay(IN := FALSE);
				fb_CupSupply.HoldCup();
				IF bToDropcup2 THEN
					nState_Dropcup := 1;
				END_IF
			1:// dropcup
				IF fb_CupSupply.DropCup() THEN
					bDoneCupSupply := TRUE;
					bToDropcup2 := FALSE;
					nState_Dropcup := 2;
				END_IF
			2:
				fbDelay(IN := TRUE, PT := T#300MS);
				IF fbDelay.Q THEN
					nState_Dropcup := 0;
				END_IF
		END_CASE
		
		CASE nState_FoodWeight OF
			0:// waiting for transfer
				IF bDoneTransfer THEN
					fbTimer(IN := FALSE);
					i1 := i1 + 1;
					nState_FoodWeight := 1;	
				END_IF
			1:// Check cup present
				IF NOT fb_FoodWeight.bIsCupPresent THEN
					IF bypassFood THEN
						nState_FoodWeight := 3;
						bStatus_Food_order[i1] := TRUE;
					ELSE
						nState_FoodWeight := 2;
					END_IF
				ELSE
					bStatus_Food_order[i1] := FALSE;
					nState_FoodWeight := 3;
				END_IF
			2:// FoodWeight
				IF NOT fb_FoodWeight.bIsCupPresent THEN
					IF fb_FoodWeight.Auto() THEN
						bStatus_Food_order[i1] := bStatus_Food;
						nState_FoodWeight := 3;
					END_IF
				ELSE
					nState_FoodWeight := 22;
				END_IF
			22:
				fbTimer(IN := TRUE, PT := T#0.3S);
				fb_FoodWeight.Auto();
				IF fbTimer.Q THEN
					fb_FoodWeight.Init();
					nState_FoodWeight := 0;
				END_IF
			3:// check i
				IF i1 < 3 THEN
					nState_FoodWeight := 5;
				ELSE 
					i1 := 2;
					nState_FoodWeight := 4;
				END_IF
			4:// dao vi tri
				bStatus_Food_order[1] := bStatus_Food_order[2];
				bStatus_Food_order[2] := bStatus_Food_order[3];
				nState_FoodWeight := 5;
			5:// Done
				bDoneFoodWeight := TRUE;
				nState_FoodWeight := 10;
		END_CASE
		
		CASE nState_WormWeight OF
			0: // waiting for transfer
				IF bDoneTransfer THEN
					fbTimer(IN := FALSE);
					i2 := i2 + 1;;
					nState_WormWeight := 1;
				END_IF
			1:
				IF NOT fb_WormWeight.bIsCupPresent THEN
					nCount2 := nCount2 + 1;
					nState_WormWeight := 11;
				ELSE
					bStatus_Worm_order[i2] := FALSE;
					nState_WormWeight := 3;
				END_IF
			11: // check food
				IF bStatus_Food_order[1] THEN
					IF bypassWorm THEN
						bStatus_Worm_order[i2] := TRUE;
						nState_WormWeight := 3;
					ELSE
						nState_WormWeight := 2;
					END_IF
				ELSE
					bStatus_Worm_order[i2] := FALSE;
					nState_WormWeight := 3;
				END_IF	
			2:// WormWeight
				IF NOT fb_WormWeight.bIsCupPresent THEN
					IF fb_WormWeight.Auto() THEN
						bStatus_Worm_order[i2] := bStatus_Worm;
						nState_WormWeight := 3;
					END_IF
				ELSE
					nState_WormWeight := 22;
				END_IF
			22:
				fbTimer(IN := TRUE, PT := T#0.3S);
				fb_WormWeight.Auto();
				IF fbTimer.Q THEN
					fb_WormWeight.Init();
					nState_WormWeight := 0;
				END_IF
			3:// check i
				IF bStatus_Worm_order[i2] THEN
					nResult_true2 := nResult_true2 + 1;
				END_IF
				IF i2 < 3 THEN
					nState_WormWeight := 5;
				ELSE
					i2 := 2;
					nState_WormWeight := 4;
				END_IF
			4:// dao vi tri				
				nResult_false2	:= nCount2 - nResult_true2;
				bStatus_Worm_order[1] := bStatus_Worm_order[2];
				bStatus_Worm_order[2] := bStatus_Worm_order[3];
				nState_WormWeight 	  := 5;
			5:// Done 
				bDoneWormWeight       := TRUE;
				nState_WormWeight	  := 10;
		END_CASE
		
		CASE nState_LidSupply OF
			0:// waiting for transfer
				IF bDoneTransfer THEN
					i3 := i3 + 1;
					nState_LidSupply := 1;
				END_IF
			1:// check worm
				IF bStatus_Worm_order[1] THEN
					IF bypassLid THEN
						bStatus_Lid_order[i3] := FALSE;
						nState_LidSupply := 4;
					ELSE
						nState_LidSupply := 2;
					END_IF
				ELSE
					bStatus_Lid_order[i3] := FALSE;
					nState_LidSupply := 4;
				END_IF
			2:// take lid
				IF fb_LidSupply.TakeLid() THEN
					nState_LidSupply := 3;
				END_IF
			3:// drop lid
				IF fb_LidSupply.DropLid() THEN
					bStatus_Lid_order[i3] := TRUE;
					nState_LidSupply := 4;
				END_IF
			4:// check i
				IF i3 < 3 THEN
					nState_LidSupply := 6;
				ELSE
					i3 := 2;
					nState_LidSupply := 5;
				END_IF
			5:// dao vi tri
				bStatus_Lid_order[1] := bStatus_Lid_order[2];
				bStatus_Lid_order[2] := bStatus_Lid_order[3];
				nState_LidSupply 	 := 6;
			6:// Done
				bDoneLidSupply 		 := TRUE;
				nState_LidSupply 	 := 10;
		END_CASE
		
		CASE nState_LidClose OF
			0: // waiting for transfer
				IF bDoneTransfer THEN
					nState_LidClose := 1;
				END_IF
			1:// Check lid supply
				IF  bStatus_Lid_order[1] THEN
					nState_LidClose := 2;
				ELSE
					nState_LidClose := 3;
				END_IF
			2:// Close lid
				IF fb_LidClose.CloseLid() THEN
					nState_LidClose := 3;
				END_IF
			3://Done
				bDoneLidClose := TRUE;
				nState_LidClose := 10;
		END_CASE
		
		CASE nState_Transfer OF
			0:// waiting for Done module
				IF nDoneTransfer = 0 THEN
						nState_Transfer := 1;
				ELSIF nDoneTransfer > 0 THEN
					IF bDoneCupSupply AND bDoneFoodWeight AND bDoneWormWeight AND bDoneLidSupply AND bDoneLidClose THEN
						nState_Transfer := 1;
					END_IF
				END_IF
			1:	
				IF fb_CupSupply.isCupDrop THEN
					bDoneCupSupply 	:= FALSE;
					bDoneFoodWeight := FALSE;
					bDoneWormWeight := FALSE;
					bDoneLidSupply 	:= FALSE;
					bDoneLidClose 	:= FALSE;
					nState_Transfer := 11;
				ELSE
					F_SetError(24,nLine := 2);
				END_IF
			11:// transfer
				IF fb_Transfer.Auto() THEN
					nShoot2 := nShoot2 + 1;
					nState_Transfer:= 2;
				END_IF
			2:
				nState_FoodWeight := 0;
				nState_WormWeight := 0;
				nState_LidSupply  := 0;
				nState_LidClose	  := 0;
				nState_Transfer	  := 0;
		END_CASE
		//Stop button
		IF bStop2 THEN
			nState := 3;
			bStartLine2 := FALSE;
		ELSIF bShift_is_over2 THEN
			nState := 4;
		END_IF
	3://Stop
		bResetAuto2		:= TRUE;
		nStatus2		:= 'RUN';
		bfinish2		:= FALSE;
		IF bypassfood THEN
			fb_FoodMixer.Stop();
		ELSE
			fb_FoodMixer.Auto();
		END_IF
		CASE nState_Dropcup OF
			0:// waiting for transfer
				fbDelay(IN := FALSE);
				fb_CupSupply.HoldCup();
				IF bToDropcup2 THEN
					nState_Dropcup := 1;
				END_IF
				IF bFinishTransfer THEN
					nState_Dropcup := 10;
				END_IF
			1:// dropcup
				IF fb_CupSupply.DropCup() THEN
					bDoneCupSupply := TRUE;
					bToDropcup2 := FALSE;
					nState_Dropcup := 2;
				END_IF
			2:
				fbDelay(IN := TRUE, PT := T#300MS);
				IF fbDelay.Q THEN
					nState_Dropcup := 0;
				END_IF
			10:// finish
				bDoneCupSupply := TRUE;
				bFinishCupSupply := TRUE;
		END_CASE
		
		CASE nState_FoodWeight OF
			0:// waiting for transfer
				IF bDoneTransfer THEN
					i1 := i1 + 1;
					fbTimer(IN := FALSE);
					nState_FoodWeight := 1;	
				END_IF
			1:// Check cup present
				IF NOT fb_FoodWeight.bIsCupPresent THEN
					IF bypassFood THEN
						nState_FoodWeight := 3;
						bStatus_Food_order[i1] := TRUE;
					ELSE
						nState_FoodWeight := 2;
					END_IF
				ELSE
					bStatus_Food_order[i1] := FALSE;
					nState_FoodWeight := 3;
				END_IF
			2:// FoodWeight
				IF NOT fb_FoodWeight.bIsCupPresent THEN
					IF fb_FoodWeight.Auto() THEN
						bStatus_Food_order[i1] := bStatus_Food;
						nState_FoodWeight := 3;
					END_IF
				ELSE
					nState_FoodWeight := 22;
				END_IF
			22:
				fbTimer(IN := TRUE, PT := T#0.3S);
				fb_FoodWeight.Auto();
				IF fbTimer.Q THEN
					fb_FoodWeight.Init();
					nState_FoodWeight := 0;
				END_IF
			3:// check i
				IF i1 < 3 THEN
					nState_FoodWeight := 5;
				ELSE 
					i1 := 2;
					nState_FoodWeight := 4;
				END_IF
			4:// dao vi tri
				bStatus_Food_order[1] := bStatus_Food_order[2];
				bStatus_Food_order[2] := bStatus_Food_order[3];
				nState_FoodWeight := 5;
			5:// Done
				bDoneFoodWeight := TRUE;
				nState_FoodWeight := 10;
			10:// finish
				bFinishFoodWeight := TRUE;
		END_CASE
		
		CASE nState_WormWeight OF
			0: // waiting for transfer
				IF bDoneTransfer THEN
					fbTimer(IN := FALSE);
					i2 := i2 + 1;;
					nState_WormWeight := 1;
				END_IF
			1:
				IF NOT fb_WormWeight.bIsCupPresent THEN
					nCount2 := nCount2 + 1;
					nState_WormWeight := 11;
				ELSE
					bStatus_Worm_order[i2] := FALSE;
					nState_WormWeight := 3;
				END_IF
			11: // check food
				IF bStatus_Food_order[1] THEN
					IF bypassWorm THEN
						bStatus_Worm_order[i2] := TRUE;
						nState_WormWeight := 3;
					ELSE
						nState_WormWeight := 2;
					END_IF
				ELSE
					bStatus_Worm_order[i2] := FALSE;
					nState_WormWeight := 3;
				END_IF	
			2:// WormWeight
				IF NOT fb_WormWeight.bIsCupPresent THEN
					IF fb_WormWeight.Auto() THEN
						bStatus_Worm_order[i2] := bStatus_Worm;
						nState_WormWeight := 3;
					END_IF
				ELSE
					nState_WormWeight := 22;
				END_IF
			22:
				fbTimer(IN := TRUE, PT := T#0.3S);
				fb_WormWeight.Auto();
				IF fbTimer.Q THEN
					fb_WormWeight.Init();
					nState_WormWeight := 0;
				END_IF
			3:// check i
				IF bStatus_Worm_order[i2] THEN
					nResult_true2 := nResult_true2 + 1;
				END_IF
				IF i2 < 3 THEN
					nState_WormWeight := 5;
				ELSE
					i2 := 2;
					nState_WormWeight := 4;
				END_IF
			4:// dao vi tri
				nResult_false2 := nCount2 - nResult_true2;
				bStatus_Worm_order[1] := bStatus_Worm_order[2];
				bStatus_Worm_order[2] := bStatus_Worm_order[3];
				nState_WormWeight 	  := 5;
			5:// Done 
				bDoneWormWeight       := TRUE;
				nState_WormWeight	  := 10;
			10:// finish
				bFinishWormWeight	  := TRUE;
		END_CASE
		
		CASE nState_LidSupply OF
			0:// waiting for transfer
				IF bDoneTransfer THEN
					i3 := i3 + 1;
					nState_LidSupply := 1;
				END_IF
			1:// check worm
				IF bStatus_Worm_order[1] THEN
					IF bypassLid THEN
						bStatus_Lid_order[i3] := FALSE;
						nState_LidSupply := 4;
					ELSE
						nState_LidSupply := 2;
					END_IF
				ELSE
					bStatus_Lid_order[i3] := FALSE;
					nState_LidSupply := 4;
				END_IF
			2:// take lid
				IF fb_LidSupply.TakeLid() THEN
					nState_LidSupply := 3;
				END_IF
			3:// drop lid
				IF fb_LidSupply.DropLid() THEN
					bStatus_Lid_order[i3] := TRUE;
					nState_LidSupply := 4;
				END_IF
			4:// check i
				IF i3 < 3 THEN
					nState_LidSupply := 6;
				ELSE
					i3 := 2;
					nState_LidSupply := 5;
				END_IF
			5:// dao vi tri
				bStatus_Lid_order[1] := bStatus_Lid_order[2];
				bStatus_Lid_order[2] := bStatus_Lid_order[3];
				nState_LidSupply 	 := 6;
			6:// Done
				bDoneLidSupply 		 := TRUE;
				nState_LidSupply 	 := 10;
			10:// finish
				bFinishLidSupply	 := TRUE;
		END_CASE
		
		CASE nState_LidClose OF
			0: // waiting for transfer
				IF bDoneTransfer THEN
					nState_LidClose := 1;
				END_IF
			1:// Check lid supply
				IF  bStatus_Lid_order[1] THEN
					nState_LidClose := 2;
				ELSE
					nState_LidClose := 3;
				END_IF
			2:// Close lid
				IF fb_LidClose.CloseLid() THEN
					nState_LidClose := 3;
				END_IF
			3://Done
				bDoneLidClose   := TRUE;
				nState_LidClose := 10;
			10:// finish
				bFinishLidClose := TRUE;
		END_CASE
		
		CASE nState_Transfer OF
			0:// waiting for Done module
				IF nDoneTransfer = 0 THEN
						nState_Transfer := 10;
				ELSIF nDoneTransfer > 0 THEN
					IF bDoneCupSupply AND bDoneFoodWeight AND bDoneWormWeight AND bDoneLidSupply AND bDoneLidClose THEN
						nState_Transfer := 10;
					END_IF
				END_IF
			1:
				IF fb_CupSupply.isCupDrop THEN
					bDoneCupSupply 	:= FALSE;
					bDoneFoodWeight := FALSE;
					bDoneWormWeight := FALSE;
					bDoneLidSupply 	:= FALSE;
					bDoneLidClose 	:= FALSE;
					nState_Transfer := 11;
				ELSE 
					F_SetError(24,nLine:=2);
				END_IF
			11:// transfer
				IF fb_Transfer.Auto() THEN
					nShoot2 := nShoot2 + 1;
					nState_Transfer:= 2;
				END_IF
			2:	
				nState_FoodWeight := 0;
				nState_WormWeight := 0;
				nState_LidSupply  := 0;
				nState_LidClose	  := 0;
				nState_Dropcup 	  := 0;
				nState_Transfer := 0;
			10:// finish
				bFinishTransfer		:= TRUE;
		END_CASE
		
		IF bFinishCupSupply AND bFinishFoodWeight AND bFinishWormWeight AND bFinishLidSupply AND bFinishLidClose AND bFinishTransfer THEN
			bfinish2 := TRUE;
			nState := 11;
		END_IF
	4:// shift is over
		bResetAuto2		:= TRUE;
		IF bypassfood THEN
			fb_FoodMixer.Stop();
		ELSE
			fb_FoodMixer.Auto();
		END_IF
		fb_CupSupply.CheckCup();
		fb_LidSupply.CheckLid();
		bStatusStart2 := FALSE;
		bfinish2		:= FALSE;
		bStart2		:= FALSE;
		nStatus2	:= 'RUN';
		bDone(CLK := bDoneTransfer);
		CASE nstateCycle OF 
			0:
				fbTimerCycle(IN := TRUE, PT := T#100S);
				IF bDone.Q THEN
					nstateCycle := 1;
				END_IF
			1:
				timeCycle := TIME_TO_REAL(fbTimerCycle.ET)/1000;
				nstateCycle := 2;
			2: 
				fproduct := REAL_TO_INT(3600/(timeCycle+0.001));
				fbTimerCycle(IN := FALSE);
				nstateCycle := 0;
		END_CASE
		CASE nState_Dropcup OF
			0:// waiting for transfer
				fbDelay(IN := FALSE);
				fb_CupSupply.HoldCup();
				IF bToDropcup2 THEN
					nState_Dropcup := 10;
				END_IF
			1:// dropcup
				IF fb_CupSupply.DropCup() THEN
					bDoneCupSupply := TRUE;
					bToDropcup2 := FALSE;
					nState_Dropcup := 2;
				END_IF
			2:
				fbDelay(IN := TRUE, PT := T#300MS);
				IF fbDelay.Q THEN
					nState_Dropcup := 0;
				END_IF
			10:// finish
				bDoneCupSupply := TRUE;
				bFinishCupSupply := TRUE;
		END_CASE
		
		CASE nState_FoodWeight OF
			0:// waiting for transfer
				IF bDoneTransfer AND nDoneTransferStop < 4 THEN
					fbTimer(IN := FALSE);
					i1 := i1 + 1;
					nState_FoodWeight := 1;	
				ELSIF bDoneTransfer AND nDoneTransferStop >= 4 THEN
					fbTimer(IN := FALSE);
					i1 := i1 + 1;
					nState_FoodWeight := 33;	
				END_IF
			1:// Check cup present
				IF NOT fb_FoodWeight.bIsCupPresent THEN
					IF bypassFood THEN
						nState_FoodWeight := 3;
						bStatus_Food_order[i1] := TRUE;
					ELSE
						nState_FoodWeight := 2;
					END_IF
				ELSE
					bStatus_Food_order[i1] := FALSE;
					nState_FoodWeight := 3;
				END_IF
			2:// FoodWeight
				IF NOT fb_FoodWeight.bIsCupPresent THEN
					IF fb_FoodWeight.Auto() THEN
						bStatus_Food_order[i1] := bStatus_Food;
						nState_FoodWeight := 3;
					END_IF
				ELSE
					nState_FoodWeight := 22;
				END_IF
			22:
				fbTimer(IN := TRUE, PT := T#0.3S);
				fb_FoodWeight.Auto();
				IF fbTimer.Q THEN
					fb_FoodWeight.Init();
					nState_FoodWeight := 0;
				END_IF
			33:
				bStatus_Food_order[i1] := FALSE;
				nState_FoodWeight := 3;
			3:// check i
				IF i1 < 3 THEN
					nState_FoodWeight := 5;
				ELSE 
					i1 := 2;
					nState_FoodWeight := 4;
				END_IF
			4:// dao vi tri
				bStatus_Food_order[1] := bStatus_Food_order[2];
				bStatus_Food_order[2] := bStatus_Food_order[3];
				nState_FoodWeight := 5;
			5:// Done
				bDoneFoodWeight := TRUE;
				nState_FoodWeight := 10;
			10:// finish
				bFinishFoodWeight := TRUE;
		END_CASE
		
		CASE nState_WormWeight OF
			0: // waiting for transfer
				IF bDoneTransfer AND nDoneTransferStop < 6 THEN
					fbTimer(IN := FALSE);
					i2 := i2 + 1;;
					nState_WormWeight := 1;
				ELSIF bDoneTransfer AND nDoneTransferStop >= 6 THEN
					fbTimer(IN := FALSE);
					i2 := i2 + 1;
					nState_WormWeight := 33;
				END_IF
			1:
				IF NOT fb_WormWeight.bIsCupPresent THEN
					nCount2 := nCount2 + 1;
					nState_WormWeight := 11;
				ELSE
					bStatus_Worm_order[i2] := FALSE;
					nState_WormWeight := 3;
				END_IF
			11: // check food
				IF bStatus_Food_order[1] THEN
					IF bypassWorm THEN
						bStatus_Worm_order[i2] := TRUE;
						nState_WormWeight := 3;
					ELSE
						nState_WormWeight := 2;
					END_IF
				ELSE
					bStatus_Worm_order[i2] := FALSE;
					nState_WormWeight := 3;
				END_IF	
			2:// WormWeight
				IF NOT fb_WormWeight.bIsCupPresent THEN
					IF fb_WormWeight.Auto() THEN
						bStatus_Worm_order[i2] := bStatus_Worm;
						nState_WormWeight := 3;
					END_IF
				ELSE
					nState_WormWeight := 22;
				END_IF
			22:
				fbTimer(IN := TRUE, PT := T#0.3S);
				fb_WormWeight.Auto();
				IF fbTimer.Q THEN
					fb_WormWeight.Init();
					nState_WormWeight := 0;
				END_IF
			33:
				bStatus_Worm_order[i2] := FALSE;
				nState_WormWeight := 3;
			3:// check i
				IF bStatus_Worm_order[i2] THEN
					nResult_true2 := nResult_true2 + 1;
				END_IF
				IF i2 < 3 THEN
					nState_WormWeight := 5;
				ELSE
					i2 := 2;
					nState_WormWeight := 4;
				END_IF
			4:// dao vi tri
				nResult_false2 := nCount2 - nResult_true2;
				bStatus_Worm_order[1] := bStatus_Worm_order[2];
				bStatus_Worm_order[2] := bStatus_Worm_order[3];
				nState_WormWeight 	  := 5;
			5:// Done 
				bDoneWormWeight       := TRUE;
				nState_WormWeight	  := 10;
			10:// finish
				bFinishWormWeight	  := TRUE;
		END_CASE
		
		CASE nState_LidSupply OF
			0:// waiting for transfer
				IF bDoneTransfer THEN
					i3 := i3 + 1;
					nState_LidSupply := 1;
				END_IF
			1:// check worm
				IF bStatus_Worm_order[1] THEN
					IF bypassLid THEN
						bStatus_Lid_order[i3] := FALSE;
						nState_LidSupply := 4;
					ELSE
						nState_LidSupply := 2;
					END_IF
				ELSE
					bStatus_Lid_order[i3] := FALSE;
					nState_LidSupply := 4;
				END_IF
			2:// take lid
				IF fb_LidSupply.TakeLid() THEN
					nState_LidSupply := 3;
				END_IF
			3:// drop lid
				IF fb_LidSupply.DropLid() THEN
					bStatus_Lid_order[i3] := TRUE;
					nState_LidSupply := 4;
				END_IF
			4:// check i
				IF i3 < 3 THEN
					nState_LidSupply := 6;
				ELSE
					i3 := 2;
					nState_LidSupply := 5;
				END_IF
			5:// dao vi tri
				bStatus_Lid_order[1] := bStatus_Lid_order[2];
				bStatus_Lid_order[2] := bStatus_Lid_order[3];
				nState_LidSupply 	 := 6;
			6:// Done
				bDoneLidSupply 		 := TRUE;
				nState_LidSupply 	 := 10;
			10:// finish
				bFinishLidSupply	 := TRUE;
		END_CASE
		
		CASE nState_LidClose OF
			0: // waiting for transfer
				IF bDoneTransfer THEN
					nState_LidClose := 1;
				END_IF
			1:// Check lid supply
				IF  bStatus_Lid_order[1] THEN
					nState_LidClose := 2;
				ELSE
					nState_LidClose := 3;
				END_IF
			2:// Close lid
				IF fb_LidClose.CloseLid() THEN
					nState_LidClose := 3;
				END_IF
			3://Done
				bDoneLidClose   := TRUE;
				nState_LidClose := 10;
			10:// finish
				bFinishLidClose := TRUE;
		END_CASE
		
		CASE nState_Transfer OF
			0:// waiting for Done module
				IF bDoneCupSupply AND bDoneFoodWeight AND bDoneWormWeight AND bDoneLidSupply AND bDoneLidClose THEN
					nState_Transfer := 1;
				END_IF
			1:
				IF fb_CupSupply.isCupDrop THEN
					bDoneCupSupply 	:= FALSE;
					bDoneFoodWeight := FALSE;
					bDoneWormWeight := FALSE;
					bDoneLidSupply 	:= FALSE;
					bDoneLidClose 	:= FALSE;
					nState_Transfer := 11;
				ELSE
					F_SetError(24,nLine := 2);
				END_IF
			11:// transfer
				IF fb_Transfer.Auto() THEN
					nShoot2 := nShoot2 + 1;
					nState_Transfer:= 2;
				END_IF
			2:
				nState_FoodWeight := 0;
				nState_WormWeight := 0;
				nState_LidSupply  := 0;
				nState_LidClose	  := 0;
				nDoneTransferStop := nDoneTransferStop + 1;
				nState_Transfer   := 3;
			3:
				IF nDoneTransferStop < 11 THEN
					nState_Transfer   := 0;
				ELSE
					nState_Transfer   := 10;
				END_IF
			10:// finish
				bFinishTransfer		:= TRUE;
		END_CASE
		IF bFinishCupSupply AND bFinishFoodWeight AND bFinishWormWeight AND bFinishLidSupply AND bFinishLidClose AND bFinishTransfer THEN
			bfinish2	:= TRUE;
			nState := 0;
		END_IF
END_CASE
END_ACTION

ACTION check:
IF fb_CupSupply.fbCylinder_Up.bIsRetract THEN
	bCylinder_up_retract 	:= TRUE;
	bCylinder_up_extend		:= FALSE;
ELSE
	bCylinder_up_retract 	:= FALSE;
	bCylinder_up_extend		:= TRUE;
END_IF

IF fb_CupSupply.fbCylinder_Dw.bIsExtend THEN
	bCylinder_dw_extend 	:= TRUE;
	bCylinder_dw_retract 	:= FALSE;
ELSIF fb_CupSupply.fbCylinder_Dw.bIsRetract THEN
	bCylinder_dw_extend 	:= FALSE;
	bCylinder_dw_retract 	:= TRUE;
ELSE
	bCylinder_dw_extend 	:= FALSE;
	bCylinder_dw_retract 	:= FALSE;
END_IF

IF fb_CupSupply.fbCylinder_Suction.bIsExtend THEN
	bCylinder_Suction_cup_extend 	:= TRUE;
	bCylinder_Suction_cup_retract	:= FALSE;
ELSE
	bCylinder_Suction_cup_extend 	:= FALSE;
	bCylinder_Suction_cup_retract	:= TRUE;
END_IF

IF fb_WormWeight.fbCylinder.bIsRetract THEN
	bCylinder_Block_Worm_Extend	 := FALSE;
	bCylinder_Block_Worm_Retract := TRUE;
ELSE
	bCylinder_Block_Worm_Extend	 := TRUE;
	bCylinder_Block_Worm_Retract := FALSE;
END_IF

IF fb_LidSupply.fbCylinder_LidStopper.bIsExtend THEN
	bCylinder_LidStopper_extend 	:= TRUE;
	bCylinder_LidStopper_retract 	:= FALSE;
ELSIF fb_LidSupply.fbCylinder_LidStopper.bIsRetract THEN
	bCylinder_LidStopper_extend 	:= FALSE;
	bCylinder_LidStopper_retract 	:= TRUE;
ELSE
	bCylinder_LidStopper_extend 	:= FALSE;
	bCylinder_LidStopper_retract 	:= FALSE;
END_IF

IF fb_LidSupply.fbCylinder_Suction.bIsExtend THEN
	bCylinder_Suction_extend		:= TRUE;
	bCylinder_Suction_retract		:= FALSE;
ELSIF fb_LidSupply.fbCylinder_Suction.bIsRetract THEN
	bCylinder_Suction_extend		:= FALSE;
	bCylinder_Suction_retract		:= TRUE;
ELSE
	bCylinder_Suction_extend		:= FALSE;
	bCylinder_Suction_retract		:= FALSE;
END_IF

IF fb_LidClose.fbCylinder_LidClose.bIsExtend THEN
	bCylinder_CloseLid_Extend		:= TRUE;
	bCylinder_CloseLid_Retract		:= FALSE;
ELSIF fb_LidClose.fbCylinder_LidClose.bIsRetract THEN
	bCylinder_CloseLid_Extend		:= FALSE;
	bCylinder_CloseLid_Retract		:= TRUE;
ELSE
	bCylinder_CloseLid_Extend		:= FALSE;
	bCylinder_CloseLid_Retract		:= FALSE;
END_IF

IF fb_Transfer.fbCylinder_Comb.bIsExtend THEN
	bCylinder_Comb_Extend			:= TRUE;
	bCylinder_Comb_Retract			:= FALSE;
ELSIF fb_Transfer.fbCylinder_Comb.bIsRetract THEN
	bCylinder_Comb_Extend			:= FALSE;
	bCylinder_Comb_Retract			:= TRUE;
ELSE
	bCylinder_Comb_Extend			:= FALSE;
	bCylinder_Comb_Retract			:= FALSE;
END_IF

IF fb_Transfer.fbCylinder_Clip.bIsExtend THEN
	bCylinder_Clip_Extend			:= TRUE;
	bCylinder_Clip_Retract			:= FALSE;
ELSIF fb_Transfer.fbCylinder_Clip.bIsRetract THEN
	bCylinder_Clip_Extend			:= FALSE;
	bCylinder_Clip_Retract			:= TRUE;
ELSE
	bCylinder_Clip_Extend			:= FALSE;
	bCylinder_Clip_Retract			:= FALSE;
END_IF

IF fb_Transfer.fbCylinder_Move_Comb.bIsExtend THEN
	bCylinder_Move_Comb_Extend		:= TRUE;
	bCylinder_Move_Comb_Retract		:= FALSE;
ELSIF fb_Transfer.fbCylinder_Move_Comb.bIsRetract THEN
	bCylinder_Move_Comb_Extend		:= FALSE;
	bCylinder_Move_Comb_Retract		:= TRUE;
ELSE
	bCylinder_Move_Comb_Extend		:= FALSE;
	bCylinder_Move_Comb_Retract		:= FALSE;
END_IF

bMotor_mixer_Manual				:= FALSE;
bMotor_mixer_reverse			:= FALSE;
bMotor_Food						:= FALSE;
bMotor_Food_reverse				:= FALSE;
bMotor_vibrating_funnel			:= FALSE;
END_ACTION

ACTION Check_reset:
IF fb_CupSupply.fbCylinder_Up.bIsRetract AND fb_CupSupply.fbCylinder_Dw.bIsExtend 
	AND NOT fb_WormWeight.fbCylinder.bIsRetract AND fb_LidSupply.fbCylinder_Suction.bIsRetract 
	AND fb_LidClose.fbCylinder_LidClose.bIsRetract AND fb_Transfer.fbCylinder_Comb.bIsRetract 
	AND fb_Transfer.fbCylinder_Clip.bIsRetract AND fb_Transfer.fbCylinder_Move_Comb.bIsRetract
	AND fb_CupSupply.fbCylinder_Suction.bIsExtend THEN
		bResetmanual2 := TRUE;
ELSE 
		bResetmanual2 := FALSE;
END_IF
IF bReset THEN
	bCylinder_up_retract 	:= true;
	bCylinder_up_extend		:= FALSE;
	bCylinder_dw_extend 	:= TRUE;
	bCylinder_dw_retract 	:= FALSE;
	bCylinder_Suction_cup_retract := FALSE;
	bCylinder_Suction_cup_extend 	:= TRUE;
	bCylinder_Block_Worm_Extend	 := TRUE;
	bCylinder_Block_Worm_Retract := FALSE;
	bCylinder_Suction_extend		:= FALSE;
	bCylinder_Suction_retract		:= TRUE;
	bCylinder_CloseLid_Extend		:= FALSE;
	bCylinder_CloseLid_Retract		:= TRUE;
	bCylinder_Comb_Extend			:= FALSE;
	bCylinder_Comb_Retract			:= TRUE;
	bCylinder_Clip_Extend			:= FALSE;
	bCylinder_Clip_Retract			:= TRUE;
	IF fb_Transfer.fbCylinder_Comb.bIsRetract THEN
		bCylinder_Move_Comb_Extend		:= FALSE;
		bCylinder_Move_Comb_Retract		:= TRUE;
	END_IF
	bxa := FALSE;
END_IF
END_ACTION

ACTION Init:
fb_CupSupply.Init();
fb_FoodWeight.Init();
fb_WormWeight.Init();
fb_LidSupply.Init();
fb_LidClose.Init();
fb_Transfer.Init();

nState := 0;
nState_Dropcup := 0;
nState_FoodWeight := 0;
nState_WormWeight := 0;
nState_LidSupply := 0;
nState_LidClose := 0;
nState_Transfer := 0;

bFinishCupSupply 	:= FALSE;
bFinishFoodWeight 	:= FALSE;
bFinishWormWeight	:= FALSE;
bFinishLidSupply	:= FALSE;
bFinishLidClose		:= FALSE;
bFinishTransfer		:= FALSE;

bDoneCupSupply 		:= FALSE;
bDoneFoodWeight 	:= FALSE;
bDoneWormWeight 	:= FALSE;
bDoneLidSupply 		:= FALSE;
bDoneLidClose 		:= FALSE;
bDoneTransfer		:= false;
nDoneTransferStop	  := 0;

bStatus_Food_order[1] := FALSE;
bStatus_Worm_order[1] := FALSE;
bStatus_Lid_order[1]  := FALSE;
		
i1 		:= 0;
i2 		:= 0;
i3 		:= 0;
END_ACTION

ACTION Manual:
fb_CupSupply.Manual(bCylinder_dw_extend := bCylinder_dw_extend, bCylinder_dw_retract := bCylinder_dw_retract,
					bCylinder_up_extend := bCylinder_up_extend, bCylinder_up_retract := bCylinder_up_retract,
					bCylinder_suction_extend:= bCylinder_Suction_cup_extend, bCylinder_suction_retract := bCylinder_Suction_cup_retract);

IF bxa THEN
	IF daothucan THEN
		fb_FoodMixer.Auto();
	ELSE
		fb_FoodMixer.Stop();
	END_IF
ELSE	
	daothucan := FALSE;
	fb_FoodMixer.Manual(bDown_Motor_Mixer := bDown_Motor_Mixer, bUp_Motor_Mixer := bUp_Motor_Mixer,
					bMotor_mixer_Manual := bMotor_mixer_Manual,bMotor_mixer_reverse := bMotor_mixer_reverse);

	IF bUp_Motor_Mixer THEN
		bUp_Motor_Mixer := FALSE;
	END_IF
	
	IF bDown_Motor_Mixer THEN
		bDown_Motor_Mixer := FALSE;
	END_IF
END_IF


IF bxa THEN
	CASE nstatetest1 OF 
	0:
		IF xathucan THEN
			nstatetest1 := 1;			
		END_IF
	1:
		IF fb_FoodWeight.Auto() THEN
			nstatetest1 := 2;
		END_IF
	2: 
		xathucan := FALSE;
		nstatetest1 := 3;
	3:
		nstatetest1 := 0;
	END_CASE
ELSE
	nstatetest1 := 0;
	xathucan := FALSE;
	fb_FoodWeight.Manual(bDown_Food_Motor := bDown_Food_Motor, bUp_Food_Motor := bUp_Food_Motor,
									bMotor_Food := bMotor_Food, bZero_Loadcell_Food := bZero_Loadcell_Food, bMotor_Food_Reverse := bMotor_Food_reverse);
				
	IF bUp_Food_Motor THEN
		bUp_Food_Motor := FALSE;
	END_IF
				
	IF bDown_Food_Motor THEN
		bDown_Food_Motor := FALSE;
	END_IF
				
	IF bZero_Loadcell_Food THEN
		bZero_Loadcell_Food := FALSE;
	END_IF
END_IF

IF bxa THEN
	CASE nstatetest2 OF 
	0:
		IF xasau THEN
			nstatetest2 := 1;
		END_IF
	1:
		IF fb_WormWeight.Auto() THEN
			nstatetest2 := 2;
		END_IF
	2: 
		xasau := FALSE;
		nstatetest2 := 3;
	3:
		nstatetest2 := 0;
	END_CASE
ELSE
	xasau := FALSE;
	nstatetest2 := 0;
	fb_WormWeight.Manual(bCylinder_Block_Worm_Extend := bCylinder_Block_Worm_Extend, bCylinder_Block_Worm_Retract := bCylinder_Block_Worm_Retract,
					bDown_vibrating_funnel := bDown_vibrating_funnel, bUp_vibrating_funnel := bUp_vibrating_funnel,
					bMotor_vibrating_funnel := bMotor_vibrating_funnel, bZero_Loadcell_Worm := bZero_Loadcell_Worm);
	
	IF bUp_vibrating_funnel THEN
		bUp_vibrating_funnel := FALSE;
	END_IF
	
	IF bDown_vibrating_funnel THEN
		bDown_vibrating_funnel := FALSE;
	END_IF
	
	IF bZero_Loadcell_Worm THEN
		bZero_Loadcell_Worm := FALSE;
	END_IF
END_IF

fb_LidSupply.Manual(bCylinder_LidStopper_extend := bCylinder_LidStopper_extend, bCylinder_LidStopper_retract := bCylinder_LidStopper_retract,
					bCylinder_Suction_extend := bCylinder_Suction_extend, bCylinder_Suction_retract := bCylinder_Suction_retract,
					bCupSuctionValve := bCupSuctionValve, bLidSuctionValve := bLidSuctionValve, bBlowValve := bBlowValve);

fb_LidClose.Manual(bCylinder_CloseLid_Extend := bCylinder_CloseLid_Extend, bCylinder_CloseLid_Retract := bCylinder_CloseLid_Retract);


fb_Transfer.Manual(bCylinder_Clip_Extend := bCylinder_Clip_Extend, bCylinder_Clip_Retract := bCylinder_Clip_Retract,
				   bCylinder_Comb_Extend := bCylinder_Comb_Extend, bCylinder_Comb_Retract := bCylinder_Comb_Retract,
				   bCylinder_Move_Comb_Extend := bCylinder_Move_Comb_Extend, bCylinder_Move_Comb_Retract := bCylinder_Move_Comb_Retract);

IF fb_CupSupply.fbCylinder_Suction.bIsExtend AND fb_LidSupply.fbCylinder_Suction.bIsRetract AND fb_LidClose.fbCylinder_LidClose.bIsRetract THEN
	bCheck := TRUE;
ELSE
	bCheck := FALSE;
END_IF
END_ACTION

ACTION Reset:
fb_CupSupply.Reset();
fb_FoodMixer.Reset();
fb_FoodWeight.Reset();
fb_WormWeight.Reset();
fb_LidSupply.Reset();
fb_LidClose.Reset();
fb_Transfer.Reset();
nState := 22;
END_ACTION

ACTION Stop:
fb_FoodWeight.Stop();
fb_WormWeight.Stop();
fb_LidSupply.Stop();
fb_LidClose.Stop();
fb_Transfer.Stop();
fb_CupSupply.Stop();
bLidSuctionValve		:= FALSE;
bCupSuctionValve		:= FALSE;
bResetAuto2		:= FALSE;
fb_FoodMixer.Stop();
END_ACTION

END_PROGRAM

// ---- POUs/Recipe/PRG_MainRecipe1.TcPOU
PROGRAM PRG_MainRecipe1
VAR
	fbrecipe		: RecipeManCommands;
	NameSave		: STRING;
	NameLoad		: STRING;
	RecipeName		: STRING;
	RecipeNameIdx	: INT;
	r1				: INT;
	dLen			: INT;
	RecipeList 		: ARRAY[0..99] OF STRING;
	tTimer			: TON;
END_VAR

PRG_RecipeList1();

FOR r1 := 0 TO 99 DO
	dLen 			:= LEN(PRG_RecipeList1.filesList[r1].sFileName) - LEN('.Recipes_1.txtrecipe'); 
	RecipeList[r1] 	:= MID(PRG_RecipeList1.filesList[r1].sFileName,dLen,1);
END_FOR

IF bSave1 THEN
	fbRecipe.CreateRecipe('Recipes_1',NameSave);
	PRG_RecipeList1.bFirst	:= TRUE;
	bSave1 					:= FALSE;
ELSIF bLoad1 THEN
	RecipeName				:= RecipeList[RecipeNameIdx];
	fbRecipe.WriteRecipe('Recipes_1', RecipeName);
	PRG_RecipeList1.bFirst	:= TRUE;
	bLoad1 					:= FALSE;
ELSIF bDelete1 THEN
	RecipeName				:= RecipeList[RecipeNameIdx];
	fbRecipe.DeleteRecipe('Recipes_1', RecipeName);		
	PRG_RecipeList1.bFirst	:= TRUE;
	bDelete1 				:= FALSE;
END_IF

END_PROGRAM

// ---- POUs/Recipe/PRG_RecipeList1.TcPOU
PROGRAM PRG_RecipeList1
VAR_INPUT
		bFirst			: BOOL := TRUE;
END_VAR
VAR
	fbEnum				: FB_EnumFindFileList;
	filesList 			: ARRAY[0..99]  OF ST_FindFileEntry;
	bNext				: BOOL;
	bAbort				: BOOL;
	bBusy				: BOOL;
	bError				: BOOL;
	nErrID				: UDINT;
	bEOE				: BOOL;
	nFindFiles			: UDINT;
END_VAR

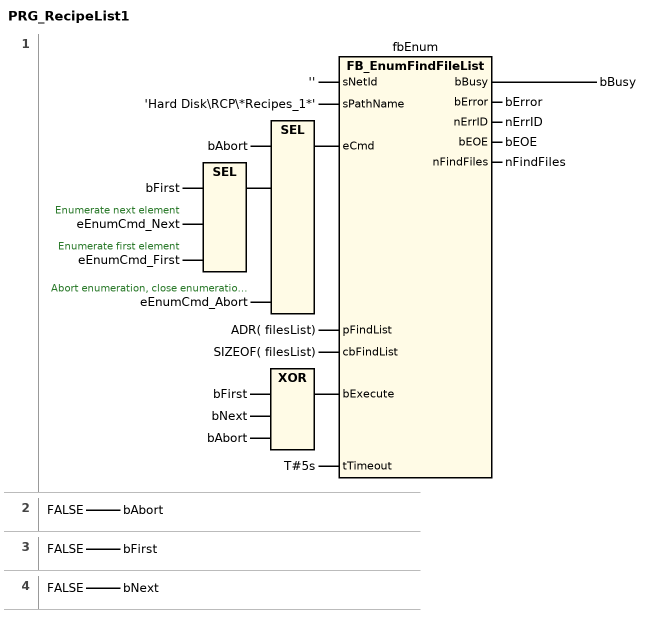
// NETWORK 1
//   eEnumCmd_Next: Enumerate next element
//   eEnumCmd_First: Enumerate first element
//   eEnumCmd_Abort: Abort enumeration, close enumeration handle.
fbEnum(
    sNetId := '',
    sPathName := 'Hard Disk\RCP\*Recipes_1*',
    eCmd := SEL(bAbort, SEL(bFirst, eEnumCmd_Next, eEnumCmd_First), eEnumCmd_Abort),
    pFindList := ADR( filesList),
    cbFindList := SIZEOF( filesList),
    bExecute := bFirst XOR bNext XOR bAbort,
    tTimeout := T#5s,
    bError => bError,
    nErrID => nErrID,
    bEOE => bEOE,
    nFindFiles => nFindFiles); // FB_EnumFindFileList
bBusy := fbEnum.bBusy;

// NETWORK 2
bAbort := FALSE;

// NETWORK 3
bFirst := FALSE;

// NETWORK 4
bNext := FALSE;

END_PROGRAM

// ---- POUs/MAIN_LINE2.TcPOU
PROGRAM MAIN_LINE2
VAR
	traError			: BOOL;
	traInitDone			: BOOL;
	bModeOff			: BOOL;
	bModeManual			: BOOL := TRUE;
	bModeAuto			: BOOL;
	Err_T				: R_TRIG;
	Wrn_T				: R_TRIG;
	fbtimer				: TON;
	fbTimerSirens		: TON;
	Run_T				: R_TRIG;
	Stop_T				: R_TRIG;
	k,k1				: INT;
	nState				: INT;
	nState1				: INT;
	nStateEmr			: INT;
	bFaultFlag			: BOOL;
	nstateStop			: INT;
	fbTimerStop			: TON;
	timerStop			: ton;
	timerReset			: TON;
	thne				: INT;
	nState2				: INT;
	Reset_T				: R_TRIG;
	fbEventlogger		: FB_Eventlogger;
	bWriteAlarm			: BOOL;
END_VAR

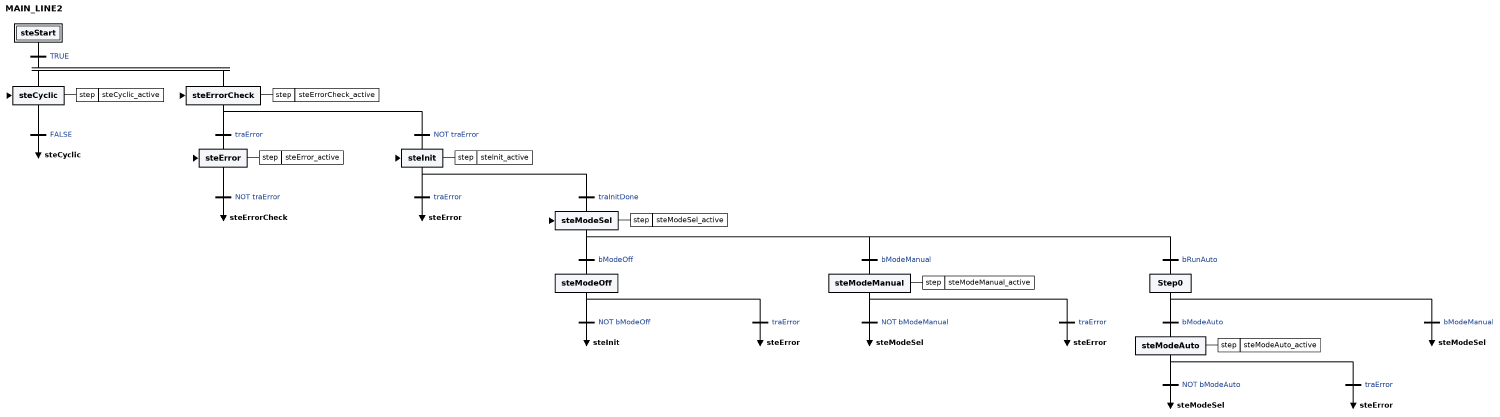
INITIAL_STEP steStart:
END_STEP
TRANSITION FROM steStart TO (steCyclic, steErrorCheck)
    := TRUE;
END_TRANSITION
STEP steCyclic:
    steCyclic_active(N);  // step action
END_STEP
TRANSITION FROM steCyclic TO steCyclic
    := FALSE;
END_TRANSITION
STEP steErrorCheck:
    steErrorCheck_active(N);  // step action
END_STEP
TRANSITION FROM steErrorCheck TO steError
    := traError;
END_TRANSITION
STEP steError:
    steError_active(N);  // step action
END_STEP
TRANSITION FROM steError TO steErrorCheck
    := NOT traError;
END_TRANSITION
TRANSITION FROM steErrorCheck TO steInit
    := NOT traError;
END_TRANSITION
STEP steInit:
    steInit_active(N);  // step action
END_STEP
TRANSITION FROM steInit TO steError
    := traError;
END_TRANSITION
TRANSITION FROM steInit TO steModeSel
    := traInitDone;
END_TRANSITION
STEP steModeSel:
    steModeSel_active(N);  // step action
END_STEP
TRANSITION FROM steModeSel TO steModeOff
    := bModeOff;
END_TRANSITION
STEP steModeOff:
END_STEP
TRANSITION FROM steModeOff TO steInit
    := NOT bModeOff;
END_TRANSITION
TRANSITION FROM steModeOff TO steError
    := traError;
END_TRANSITION
TRANSITION FROM steModeSel TO steModeManual
    := bModeManual;
END_TRANSITION
STEP steModeManual:
    steModeManual_active(N);  // step action
END_STEP
TRANSITION FROM steModeManual TO steModeSel
    := NOT bModeManual;
END_TRANSITION
TRANSITION FROM steModeManual TO steError
    := traError;
END_TRANSITION
TRANSITION FROM steModeSel TO Step0
    := bRunAuto;
END_TRANSITION
STEP Step0:
END_STEP
TRANSITION FROM Step0 TO steModeAuto
    := bModeAuto;
END_TRANSITION
TRANSITION FROM Step0 TO steModeSel
    := bModeManual;
END_TRANSITION
STEP steModeAuto:
    steModeAuto_active(N);  // step action
END_STEP
TRANSITION FROM steModeAuto TO steModeSel
    := NOT bModeAuto;
END_TRANSITION
TRANSITION FROM steModeAuto TO steError
    := traError;
END_TRANSITION

ACTION ListError:
Err_T(CLK := bError2);
Wrn_T(CLK := bWarning2);
GetLocalSystemTime(bEnable := 1,);
IF a2 > 100 THEN
	a2 := 100;
END_IF
		
CASE nState OF 
	0:
		IF Err_T.Q THEN
			nState := 1;
		ELSIF Wrn_T.Q THEN
			bWrn2 := true;
			nState := 10;
		END_IF
	1:
		CASE nErrorID OF	
			23:
				stErrorTxt2 := "E1_2.Lỗi hết hũ trạm 2 [kiểm tra U1I2-4]";
				stErrorTxt3 := 'E1_2.The jar is empty line 2 [check U1I2-4]';
				fbEventlogger(eventClass := TC_EVENTS.Entobel.Event23.uuidEventClass, nEventID := DINT_TO_UDINT(nErrorID));
			24:
				stErrorTxt2 := "E2_2.Lỗi hũ bị kẹt trạm 2 [kiểm tra U1I2-8]";
				stErrorTxt3 := 'E2_2.The jar  is trapped line 2 [check U1I2-8]';
				fbEventlogger(eventClass := TC_EVENTS.Entobel.Event24.uuidEventClass, nEventID := DINT_TO_UDINT(nErrorID));
			25:
				stErrorTxt2 := "E3_2.Lỗi ben chặn hũ trên rút về trạm 2 [kiểm tra U1I2-5]" ;
				stErrorTxt3 := 'E3_2.The upper cylinder retract  is faulty line 2 [check U1I2-5]';
				fbEventlogger(eventClass := TC_EVENTS.Entobel.Event25.uuidEventClass, nEventID := DINT_TO_UDINT(nErrorID));
			26:
				stErrorTxt2 := "E4_2.Lỗi ben chặn hũ dưới rút về trạm 2 [kiểm tra U1I2-6]";
				stErrorTxt3 := 'E4_2.The lower cylinder retract  is faulty line 2 [check U1I2-6]';
				fbEventlogger(eventClass := TC_EVENTS.Entobel.Event26.uuidEventClass, nEventID := DINT_TO_UDINT(nErrorID));
			27:
				stErrorTxt2 := "E5_2.Lỗi ben chặn hũ dưới đẩy ra trạm 2 [kiểm tra U1I2-7]";
				stErrorTxt3 := 'E5_2.The lower cylinder extend  is faulty line 2 [check U1I2-7]';
				fbEventlogger(eventClass := TC_EVENTS.Entobel.Event27.uuidEventClass, nEventID := DINT_TO_UDINT(nErrorID));
			28:
				stErrorTxt2 := "E6_2.Lỗi biến tần đảo thức ăn trạm 2 [kiểm tra biến tần 1]";
				stErrorTxt3 := 'E6_2.The inverter of agitator motor fault line 2 [check inverter 1]';
				fbEventlogger(eventClass := TC_EVENTS.Entobel.Event28.uuidEventClass, nEventID := DINT_TO_UDINT(nErrorID));
			29:
				stErrorTxt2 := "E7_2.Lỗi driver chia thức ăn trạm 2 [kiểm tra driver 1]";
				stErrorTxt3 := 'E7_2.The driver of dispenser motor fault line 2 [check driver 1]';
				fbEventlogger(eventClass := TC_EVENTS.Entobel.Event29.uuidEventClass, nEventID := DINT_TO_UDINT(nErrorID));
			30:
				stErrorTxt2 := "E8_2.Lỗi ben chặn sâu rút về trạm 2 [kiểm tra U1I3-1]";
				stErrorTxt3 := 'E8_2.The cylinder blocking worm retract is faulty line 2 [check U1I3-1]';
				fbEventlogger(eventClass := TC_EVENTS.Entobel.Event30.uuidEventClass, nEventID := DINT_TO_UDINT(nErrorID));
			31:
				stErrorTxt2 := "E9_2.Lỗi biến tần phểu rung sâu trạm 2 [kiểm tra biến tần 2]";
				stErrorTxt3 := 'E9_2.The inverter of vibrating funnel fault line 2 [check inverter 2]';
				fbEventlogger(eventClass := TC_EVENTS.Entobel.Event31.uuidEventClass, nEventID := DINT_TO_UDINT(nErrorID));
			32:
				stErrorTxt2 := "E10_2.Lỗi hết nắp trạm 2 [kiểm tra U1I3-2]";
				stErrorTxt3 := 'E10_2.The lid is empty line 2 [check U1I3-2]';
				fbEventlogger(eventClass := TC_EVENTS.Entobel.Event32.uuidEventClass, nEventID := DINT_TO_UDINT(nErrorID));
			33:
				stErrorTxt2 := "E11_2.Lỗi ben chặn nắp rút về trạm 2 [kiểm tra U1I3-3]";
				stErrorTxt3 := 'E11_2.The cylinder blocking the lid retract is faulty line 2 [check U1I3-3]';
				fbEventlogger(eventClass := TC_EVENTS.Entobel.Event33.uuidEventClass, nEventID := DINT_TO_UDINT(nErrorID));
			34:
				stErrorTxt2 := "E12_2.Lỗi ben chặn nắp đẩy ra trạm 2 [kiểm tra U1I3-4]";
				stErrorTxt3 := 'E12_2.The cylinder blocking the lid extend is faulty line 2 [check U1I3-4]';
				fbEventlogger(eventClass := TC_EVENTS.Entobel.Event34.uuidEventClass, nEventID := DINT_TO_UDINT(nErrorID));
			35:
				stErrorTxt2 := "E13_2.Lỗi ben hút/thả nắp rút ra trạm 2 [kiểm tra U1I3-5]";
				stErrorTxt3 := 'E13_2.The cylinder sucking the lid retract is faulty line 2 [check U1I3-5]';
				fbEventlogger(eventClass := TC_EVENTS.Entobel.Event35.uuidEventClass, nEventID := DINT_TO_UDINT(nErrorID));
			36:
				stErrorTxt2 := "E14_2.Lỗi ben hút/thả nắp đẩy ra trạm 2 [kiểm tra U1I3-6]";
				stErrorTxt3 := 'E14_2.The cylinder sucking the lid extend is faulty line 2 [check U1I3-6]';
				fbEventlogger(eventClass := TC_EVENTS.Entobel.Event36.uuidEventClass, nEventID := DINT_TO_UDINT(nErrorID));
			37:
				stErrorTxt2 := "E15_2.Lỗi ben dập nắp rút về trạm 2 [kiểm tra U1I3-8]";
				stErrorTxt3 := 'E15_2.The cylinder pressing the lid retract is faulty line 2 [check U1I3-8]';
				fbEventlogger(eventClass := TC_EVENTS.Entobel.Event37.uuidEventClass, nEventID := DINT_TO_UDINT(nErrorID));
			38:
				stErrorTxt2 := "E16_2.Lỗi ben dập nắp đẩy ra trạm 2 [kiểm tra U1I4-1]";
				stErrorTxt3 := 'E16_2.The cylinder pressing the lid extend is faulty line 2 [check U1I4-1]';
				fbEventlogger(eventClass := TC_EVENTS.Entobel.Event38.uuidEventClass, nEventID := DINT_TO_UDINT(nErrorID));
			39:
				stErrorTxt2 := "E17_2.Lỗi ben lượt ra/vào Rút về trạm 2 [kiểm tra U1I4-2]";
				stErrorTxt3 := 'E17_2.The comb cylinder retract is faulty line 2 [check U1I4-2]';
				fbEventlogger(eventClass := TC_EVENTS.Entobel.Event39.uuidEventClass, nEventID := DINT_TO_UDINT(nErrorID));
			40:
				stErrorTxt2 := "E18_2.Lỗi ben lượt ra/vào đẩy ra trạm 2 [kiểm tra U1I4-3]";
				stErrorTxt3 := 'E18_2.The comb cylinder extend is faulty line 2 [check U1I4-3]';
				fbEventlogger(eventClass := TC_EVENTS.Entobel.Event40.uuidEventClass, nEventID := DINT_TO_UDINT(nErrorID));
			41:
				stErrorTxt2 := "E19_2.Lỗi ben kẹp hũ rút về trạm 2 [kiểm tra U1I4-6]";
				stErrorTxt3 := 'E19_2.The clap cylinder retract is faulty line 2 [check U1I4-6]';
				fbEventlogger(eventClass := TC_EVENTS.Entobel.Event41.uuidEventClass, nEventID := DINT_TO_UDINT(nErrorID));
			42:
				stErrorTxt2 := "E20_2.Lỗi ben kẹp hũ đẩy ra trạm 2 [kiểm tra U1I4-7]";	
				stErrorTxt3 := 'E20_2.The clap cylinder extend is faulty 2 [check U1I4-4]';
				fbEventlogger(eventClass := TC_EVENTS.Entobel.Event42.uuidEventClass, nEventID := DINT_TO_UDINT(nErrorID));
			43:
				stErrorTxt2 := "E21_2.Lỗi ben di chuyển lượt rút về trạm 2 [kiểm tra U1I4-4]";	
				stErrorTxt3 := 'E21_2.The cylinder moving comb retract is faulty line 2 [check U1I4-4]';
				fbEventlogger(eventClass := TC_EVENTS.Entobel.Event43.uuidEventClass, nEventID := DINT_TO_UDINT(nErrorID));
			44:
				stErrorTxt2 := "E22_2.Lỗi ben di chuyển lượt đẩy ra trạm 2 [kiểm tra U1I4-5]";	
				stErrorTxt3 := 'E22_2.The cylinder moving comb extend is faulty line 2 [check U1I4-5]';
				fbEventlogger(eventClass := TC_EVENTS.Entobel.Event44.uuidEventClass, nEventID := DINT_TO_UDINT(nErrorID));
			46:
				stErrorTxt2 := "E23_2.Lỗi mất hũ khi đang cân thức ăn trạm 2 [kiểm tra U1I4-8]";
				stErrorTxt3 := 'E23_2.The jar is missed when weighting food line 2 [check U1I4-8]';
				fbEventlogger(eventClass := TC_EVENTS.Entobel.Event46.uuidEventClass, nEventID := DINT_TO_UDINT(nErrorID));
			48:
				stErrorTxt2 := "E24_2.Lỗi mất hũ khi đang cân sâu trạm 2 [kiểm tra U1I5-1]";
				stErrorTxt3 := 'E24_2.The jar is missed when weighting larvae line 2 [check U1I5-1]';
				fbEventlogger(eventClass := TC_EVENTS.Entobel.Event48.uuidEventClass, nEventID := DINT_TO_UDINT(nErrorID));
			50:
				stErrorTxt2 := "E25_2.Lỗi hút không được nắp trạm 2 [kiểm tra U1I3-7]";
				stErrorTxt3 := 'E25_2.Failed to suction the lid  line 2 [check U1I3-7]';
				fbEventlogger(eventClass := TC_EVENTS.Entobel.Event50.uuidEventClass, nEventID := DINT_TO_UDINT(nErrorID));
			52:
				stErrorTxt2 := "E26_2.Lỗi nắp đã được hút 2 [kiểm tra U1I3-7]";	
				stErrorTxt3 := 'E26_2.The lid is still on the valve line 2 [check U1I3-7]';
				fbEventlogger(eventClass := TC_EVENTS.Entobel.Event52.uuidEventClass, nEventID := DINT_TO_UDINT(nErrorID));
			53:
				stErrorTxt2 := "E27_2.Lỗi an toàn cửa 1 [kiểm tra U1I7-8]";	
				stErrorTxt3 := 'E27_2.The safety door 1 is error [check U1I7-8]';
			54:
				stErrorTxt2 := "E28_2.Lỗi an toàn cửa 2 [kiểm tra U1I7-9]";
				stErrorTxt3 := 'E28_2.The safety door 2 is error [check U1I7-9]';
			55:
				stErrorTxt2 := "E29_2.Lỗi an toàn cửa 3 [kiểm tra U1I7-10]";
				stErrorTxt3 := 'E29_2.The safety door 3 is error [check U1I7-10]';
			58: 
				stErrorTxt2 := "E30_2.Lỗi quá cân thức ăn trạm 2 [kiểm tra cân thức ăn]";
				stErrorTxt3 := 'E30_2.Overload weightfood line 2 [check weightfood]';
				fbEventlogger(eventClass := TC_EVENTS.Entobel.Event58.uuidEventClass, nEventID := DINT_TO_UDINT(nErrorID));
			59: 
				stErrorTxt2 := "E31_2.Lỗi quá cân sâu trạm 2 [kiểm tra cân sâu]";
				stErrorTxt3 := 'E31_2.Overload weightlarvae line 2 [check weightlarvae]';
				fbEventlogger(eventClass := TC_EVENTS.Entobel.Event59.uuidEventClass, nEventID := DINT_TO_UDINT(nErrorID));
			61:
				stErrorTxt2 := "E32_2.Lỗi ben hút/thả hũ đẩy ra trạm 2 [kiểm tra U1I7-12]";
				stErrorTxt3 := 'E32_2.The cylinder sucking the jar is faulty line 2 [check U1I7-12]';
				fbEventlogger(eventClass := TC_EVENTS.Entobel.Event61.uuidEventClass, nEventID := DINT_TO_UDINT(nErrorID));
			62:
				stErrorTxt2 := "E33_2.Lỗi Modbus thiết bị 1";
				stErrorTxt3 := 'E33_2.Error Modbus device 1';
				fbEventlogger(eventClass := TC_EVENTS.Entobel.Event62.uuidEventClass, nEventID := DINT_TO_UDINT(nErrorID));
			63:
				stErrorTxt2 := "E34_2.Lỗi Modbus thiết bị 2";
				stErrorTxt3 := 'E34_2.Error Modbus device 2';
				fbEventlogger(eventClass := TC_EVENTS.Entobel.Event63.uuidEventClass, nEventID := DINT_TO_UDINT(nErrorID));
			64:
				stErrorTxt2 := "E35_2.Lỗi Modbus thiết bị 3";
				stErrorTxt3 := 'E35_2.Error Modbus device 3';
			67:
				stErrorTxt2 := "E36_2.Lỗi Modbus thiết bị 6";
				stErrorTxt3 := 'E36_2.Error Modbus device 6';
				fbEventlogger(eventClass := TC_EVENTS.Entobel.Event67.uuidEventClass, nEventID := DINT_TO_UDINT(nErrorID));
			71:
				stErrorTxt2 := "E37_2.Lỗi đầu cân thức ăn Laumas";
				stErrorTxt3 := 'E37_2.Error Laumas 1';
				fbEventlogger(eventClass := TC_EVENTS.Entobel.Event71.uuidEventClass, nEventID := DINT_TO_UDINT(nErrorID));
			72:
				stErrorTxt2 := "E38_2.Lỗi đầu cân sâu Laumas";
				stErrorTxt3 := 'E38_2.Error Laumas 2';
				fbEventlogger(eventClass := TC_EVENTS.Entobel.Event72.uuidEventClass, nEventID := DINT_TO_UDINT(nErrorID));
			74:
				stErrorTxt2 := "E39_2.Lỗi ben chặn sâu đẩy ra trạm 2 [kiểm tra U1I3-1]";
				stErrorTxt3 := 'E39_2.The cylinder blocking worm extend  is faulty line 2';
				fbEventlogger(eventClass := TC_EVENTS.Entobel.Event74.uuidEventClass, nEventID := DINT_TO_UDINT(nErrorID));
			75:
				stErrorTxt2 := "E40_2.Lỗi thiếu khí đầu vào [kiểm tra U1I7-13]";
				stErrorTxt3 := 'E40_2.Error of lack of input air [check U1I7-13]';	
			78:
				stErrorTxt2 := "E41_2.Lỗi hết thức ăn trạm 2";
				stErrorTxt3 := 'E41_2.Error running out of food line 2';
				fbEventlogger(eventClass := TC_EVENTS.Entobel.Event77.uuidEventClass, nEventID := DINT_TO_UDINT(nErrorID));	
			79:
				stErrorTxt2 := "E42_2.Lỗi hết sâu trạm 2";
				stErrorTxt3 := 'E42_2.Error running out of larvae line 2';
				fbEventlogger(eventClass := TC_EVENTS.Entobel.Event79.uuidEventClass, nEventID := DINT_TO_UDINT(nErrorID));	
			98:
				stErrorTxt2 := "E98_2.Dừng khẩn [kiểm tra Emergency]"; 
				stErrorTxt3 := 'E98_2.Emergency Stop [check Emergency]';
			99: 
				stErrorTxt2 := "E99_2.Lỗi biến tần băng tải đầu ra [kiểm tra biến tần 3]";
				stErrorTxt3 := 'E99_2.The inverter of conveyor ouy [check inverter 3]';
		END_CASE
		IF a2 <> 1 THEN
			FOR	k := a2 TO 2 BY -1 DO
				nErrorIDList2[k].nErrorID 	 := nErrorIDList2[k-1].nErrorID;
				nErrorIDList2[k].ErrorTime   := nErrorIDList2[k-1].ErrorTime;
				nErrorIDList2[k].ErrorStatus := nErrorIDList2[k-1].ErrorStatus;	
			END_FOR		
		END_IF 
		nErrorIDList2[1].nErrorID := nErrorID;
		nErrorIDList2[1].ErrorTime := SYSTEMTIME_TO_DT(GetLocalSystemTime.systemTime);
		nErrorIDList2[1].ErrorStatus := 1;
		nStatus2	:= 'ERROR';
		a2 := a2 + 1;
		bWarning := FALSE;
		nState := 2;
	2:
		bWriteAlarm	:= TRUE;
		IF nErrorID = 53 THEN
			bTo_alarm_side2 := FALSE;
		ELSIF nErrorID = 54 THEN
			bTo_alarm_side2 := FALSE;
		ELSIF nErrorID = 55 THEN
			bTo_alarm_side2 := FALSE;
		ELSIF nErrorID = 64 THEN
			bTo_alarm_side2 := FALSE;
		ELSIF nErrorID = 75 THEN
			bTo_alarm_side2 := FALSE;
		ELSIF nErrorID = 98 THEN
			bTo_alarm_side2 := FALSE;
		ELSIF nErrorID = 99 THEN
			bTo_alarm_side2 := FALSE;
		ELSE 	
			bTo_alarm_side2 := TRUE;
		END_IF
		bSirens := TRUE;
		nState := 3;
	3:
		IF NOT bError2 THEN
			nState 	:= 0;
		END_IF
	10:
		CASE nWarningID OF
			108:
				stWarningTxt2 := "W1_2.Cảnh báo hết hũ trạm 2 [kiểm tra U1I2-4]";
				stWarningTxt3 := 'W1_2.Warning out of jar line 2 [check U1I2-4]';
				fbEventlogger(eventClass := TC_EVENTS.Entobel.Event108.uuidEventClass, nEventID := DINT_TO_UDINT(nWarningID));
			109:
				stWarningTxt2 := "W2_2.Cảnh báo hết nắp trạm 2 [kiểm tra U1I3-2]";
				stWarningTxt3 := 'W2_2.Warning out of lid line 2 [check U1I3-2]';
				fbEventlogger(eventClass := TC_EVENTS.Entobel.Event109.uuidEventClass, nEventID := DINT_TO_UDINT(nWarningID));
			110:
				stWarningTxt2 := "W3_2.Cảnh báo hết thức ăn trạm 2";
				stWarningTxt3 := 'W3_2.Warning running out of food line 2';
				fbEventlogger(eventClass := TC_EVENTS.Entobel.Event110.uuidEventClass, nEventID := DINT_TO_UDINT(nWarningID));
			111:
				stWarningTxt2 := "W4_2.Cảnh báo cân quá khối lượng thức ăn trạm 2";
				stWarningTxt3 := 'W4_2.Warning food weight exceeds limit line 2';
				fbEventlogger(eventClass := TC_EVENTS.Entobel.Event111.uuidEventClass, nEventID := DINT_TO_UDINT(nWarningID));
			112:
				stWarningTxt2 := "W5_2.Cảnh báo hết sâu trạm 2";
				stWarningTxt3 := 'W5_2.Warning running out of larvae line 2';
				fbEventlogger(eventClass := TC_EVENTS.Entobel.Event112.uuidEventClass, nEventID := DINT_TO_UDINT(nWarningID));
			113:
				stWarningTxt2 := "W6_2.Canh bao can qua khoi luong sau tram 2";
				stWarningTxt3 := 'W6_2.Warning larvae weight exceeds limit line 2';
				fbEventlogger(eventClass := TC_EVENTS.Entobel.Event113.uuidEventClass, nEventID := DINT_TO_UDINT(nWarningID));
			114:
				stWarningTxt2 := "W7_2.Cảnh báo dập nắp không vô trạm 2 [kiểm tra U1I4-1]";
				stWarningTxt3 := 'W7_2.Warning do not press lid inward line 2 [check U1I4-1]';
				fbEventlogger(eventClass := TC_EVENTS.Entobel.Event114.uuidEventClass, nEventID := DINT_TO_UDINT(nWarningID));
			115:
				stWarningTxt2 := "W8_2.Cảnh báo mất kết nối với PC Advantech [kiểm tra PC]";
				stWarningTxt3 := 'W8_2.Warning disconnect to PC Advantech [check PC]';	
		END_CASE
		IF a2 <> 1 THEN
			FOR	k := a2 TO 2 BY -1 DO
				nErrorIDList2[k].nErrorID 	 := nErrorIDList2[k-1].nErrorID;
				nErrorIDList2[k].ErrorTime   := nErrorIDList2[k-1].ErrorTime;
				nErrorIDList2[k].ErrorStatus := nErrorIDList2[k-1].ErrorStatus;			
			END_FOR		
		END_IF 
		nErrorIDList2[1].nErrorID := nWarningID;
		nErrorIDList2[1].ErrorTime := SYSTEMTIME_TO_DT(GetLocalSystemTime.systemTime);
		nErrorIDList2[1].ErrorStatus := 1;
		nStatus1	:= 'WARNING';
		a2 := a2 + 1;
		nState := 11;
	11:
		bWriteAlarm	:= TRUE;
		bSirens := TRUE;
		nState := 12;
	12:
		bWarning2 := FALSE;
		nState := 0;		
END_CASE

IF bclearall THEN
	FOR k := 1 TO 100 DO
		AlarmList2[1,k] := "";
		AlarmList2[2,k] := "";	
		AlarmList2[3,k] := "";
		AlarmList2[4,k] := "";	
		AlarmList4[1,k] := '';
		AlarmList4[2,k] := '';	
		AlarmList4[3,k] := '';
		AlarmList4[4,k] := '';	
	END_FOR
	a2 := 1;
END_IF
END_ACTION

ACTION Reset_active:
PR_Line02.Reset();
END_ACTION

ACTION steCyclic_active:
PR_Line02();
ListError();;
GetLocalSystemTime(bEnable := 1,);
SystemTimeFull 	:= SYSTEMTIME_TO_STRING(in := GetLocalSystemTime.systemTime);
PRG_MainRecipe1_1();

IF bError2 THEN
	traError := true;
END_IF

IF NOT bEmer THEN
	traError := TRUE;
END_IF
IF bWriteAlarm	THEN
FOR k1 := 1 TO 100 DO
	AlarmList2[1,k1] 	:= INT_TO_WSTRING(nErrorIDList2[k1].nErrorID);
	AlarmList4[1,k1]	:= INT_TO_STRING(nErrorIDList2[k1].nErrorID);
	AlarmList2[4,k1] 	:= STRING_TO_WSTRING(MID(STR := DT_TO_STRING(nErrorIDList2[k1].ErrorTime),LEN := 19, POS := 4));
	AlarmList4[4,k1] 	:= MID(STR := DT_TO_STRING(nErrorIDList2[k1].ErrorTime),LEN := 19, POS := 4);
	IF nErrorIDList2[k1].ErrorStatus = 1 THEN
		AlarmList2[3,k1] := "Active";
		AlarmList4[3,k1] := 'Active';
	ELSE
		AlarmList2[3,k1] := "Release";
		AlarmList4[3,k1] := 'Release';
	END_IF
	CASE nErrorIDList2[k1].nErrorID OF 
			0:
				AlarmList2[4,k1] 	:= "";
				AlarmList2[3,k1] 	:= "";
				AlarmList4[4,k1] 	:= '';
				AlarmList4[3,k1] 	:= '';
			23:
				AlarmList2[2,k1] := "E1_2.Lỗi hết hũ trạm 2 [kiểm tra U1I2-4]";
				AlarmList4[2,k1] := 'E1_2.The jar is empty line 2 [check U1I2-4]';
			24:
				AlarmList2[2,k1] := "E2_2.Lỗi hũ bị kẹt trạm 2 [kiểm tra U1I2-8]";
				AlarmList4[2,k1] := 'E2_2.The jar  is trapped line 2 [check U1I2-8]';
			25:
				AlarmList2[2,k1] := "E3_2.Lỗi ben chặn hũ trên rút về trạm 2 [kiểm tra U1I2-5]" ;
				AlarmList4[2,k1] := 'E3_2.The upper cylinder retract  is faulty line 2 [check U1I2-5]';
			26:
				AlarmList2[2,k1] := "E4_2.Lỗi ben chặn hũ dưới rút về trạm 2 [kiểm tra U1I2-6]";
				AlarmList4[2,k1] := 'E4_2.The lower cylinder retract  is faulty line 2 [check U1I2-6]';
			27:
				AlarmList2[2,k1] := "E5_2.Lỗi ben chặn hũ dưới đẩy ra trạm 2 [kiểm tra U1I2-7]";
				AlarmList4[2,k1] := 'E5_2.The lower cylinder extend  is faulty line 2 [check U1I2-7]';
			28:
				AlarmList2[2,k1] := "E6_2.Lỗi biến tần đảo thức ăn trạm 2 [kiểm tra biến tần 1]";
				AlarmList4[2,k1] := 'E6_2.The inverter of agitator motor fault line 2 [check inverter 1]';
			29:
				AlarmList2[2,k1] := "E7_2.Lỗi driver chia thức ăn trạm 2 [kiểm tra driver 1]";
				AlarmList4[2,k1] := 'E7_2.The driver of dispenser motor fault line 2 [check driver 1]';
			30:
				AlarmList2[2,k1] := "E8_2.Lỗi ben chặn sâu rút về trạm 2 [kiểm tra U1I3-1]";
				AlarmList4[2,k1] := 'E8_2.The cylinder blocking worm retract is faulty line 2 [check U1I3-1]';
			31:
				AlarmList2[2,k1] := "E9_2.Lỗi biến tần phểu rung sâu trạm 2 [kiểm tra biến tần 2]";
				AlarmList4[2,k1] := 'E9_2.The inverter of vibrating funnel fault line 2 [check inverter 2]';
			32:
				AlarmList2[2,k1] := "E10_2.Lỗi hết nắp trạm 2 [kiểm tra U1I3-2]";
				AlarmList4[2,k1] := 'E10_2.The lid is empty line 2 [check U1I3-2]';
			33:
				AlarmList2[2,k1] := "E11_2.Lỗi ben chặn nắp rút về trạm 2 [kiểm tra U1I3-3]";
				AlarmList4[2,k1] := 'E11_2.The cylinder blocking the lid retract is faulty line 2 [check U1I3-3]';
			34:
				AlarmList2[2,k1] := "E12_2.Lỗi ben chặn nắp đẩy ra trạm 2 [kiểm tra U1I3-4]";
				AlarmList4[2,k1] := 'E12_2.The cylinder blocking the lid extend is faulty line 2 [check U1I3-4]';
			35:
				AlarmList2[2,k1] := "E13_2.Lỗi ben hút/thả nắp rút ra trạm 2 [kiểm tra U1I3-5]";
				AlarmList4[2,k1] := 'E13_2.The cylinder sucking the lid retract is faulty line 2 [check U1I3-5]';
			36:
				AlarmList2[2,k1] := "E14_2.Lỗi ben hút/thả nắp đẩy ra trạm 2 [kiểm tra U1I3-6]";
				AlarmList4[2,k1] := 'E14_2.The cylinder sucking the lid extend is faulty line 2 [check U1I3-6]';
			37:
				AlarmList2[2,k1] := "E15_2.Lỗi ben dập nắp rút về trạm 2 [kiểm tra U1I3-8]";
				AlarmList4[2,k1] := 'E15_2.The cylinder pressing the lid retract is faulty line 2 [check U1I3-8]';
			38:
				AlarmList2[2,k1] := "E16_2.Lỗi ben dập nắp đẩy ra trạm 2 [kiểm tra U1I4-1]";
				AlarmList4[2,k1] := 'E16_2.The cylinder pressing the lid extend is faulty line 2 [check U1I4-1]';
			39:
				AlarmList2[2,k1] := "E17_2.Lỗi ben lượt ra/vào Rút về trạm 2 [kiểm tra U1I4-2]";
				AlarmList4[2,k1] := 'E17_2.The comb cylinder retract is faulty line 2 [check U1I4-2]';
			40:
				AlarmList2[2,k1] := "E18_2.Lỗi ben lượt ra/vào đẩy ra trạm 2 [kiểm tra U1I4-3]";
				AlarmList4[2,k1] := 'E18_2.The comb cylinder extend is faulty line 2 [check U1I4-3]';
			41:
				AlarmList2[2,k1] := "E19_2.Lỗi ben kẹp hũ rút về trạm 2 [kiểm tra U1I4-6]";
				AlarmList4[2,k1] := 'E19_2.The clap cylinder retract is faulty line 2 [check U1I4-6]';
			42:
				AlarmList2[2,k1] := "E20_2.Lỗi ben kẹp hũ đẩy ra trạm 2 [kiểm tra U1I4-7]";	
				AlarmList4[2,k1] := 'E20_2.The clap cylinder extend is faulty 2 [check U1I4-4]';
			43:
				AlarmList2[2,k1] := "E21_2.Lỗi ben di chuyển lượt rút về trạm 2 [kiểm tra U1I4-4]";	
				AlarmList4[2,k1] := 'E21_2.The cylinder moving comb retract is faulty line 2 [check U1I4-4]';
			44:
				AlarmList2[2,k1] := "E22_2.Lỗi ben di chuyển lượt đẩy ra trạm 2 [kiểm tra U1I4-5]";	
				AlarmList4[2,k1] := 'E22_2.The cylinder moving comb extend is faulty line 2 [check U1I4-5]';
			46:
				AlarmList2[2,k1] := "E23_2.Lỗi mất hũ khi đang cân thức ăn trạm 2 [kiểm tra U1I4-8]";
				AlarmList4[2,k1] := 'E23_2.The jar is missed when weighting food line 2 [check U1I4-8]';
			48:
				AlarmList2[2,k1] := "E24_2.Lỗi mất hũ khi đang cân sâu trạm 2 [kiểm tra U1I5-1]";
				AlarmList4[2,k1] := 'E24_2.The jar is missed when weighting larvae line 2 [check U1I5-1]';
			50:
				AlarmList2[2,k1] := "E25_2.Lỗi hút không được nắp trạm 2 [kiểm tra U1I3-7]";
				AlarmList4[2,k1] := 'E25_2.Failed to suction the lid  line 2 [check U1I3-7]';
			52:
				AlarmList2[2,k1] := "E26_2.Lỗi nắp đã được hút 2 [kiểm tra U1I3-7]";	
				AlarmList4[2,k1] := 'E26_2.The lid is still on the valve line 2 [check U1I3-7]';
			53:
				AlarmList2[2,k1] := "E27_2.Lỗi an toàn cửa 1 [kiểm tra U1I7-8]";	
				AlarmList4[2,k1] := 'E27_2.The safety door 1 is error [check U1I7-8]';
			54:
				AlarmList2[2,k1] := "E28_2.Lỗi an toàn cửa 2 [kiểm tra U1I7-9]";
				AlarmList4[2,k1] := 'E28_2.The safety door 2 is error [check U1I7-9]';
			55:
				AlarmList2[2,k1] := "E29_2.Lỗi an toàn cửa 3 [kiểm tra U1I7-10]";
				AlarmList4[2,k1] := 'E29_2.The safety door 3 is error [check U1I7-10]';
			58: 
				AlarmList2[2,k1] := "E30_2.Lỗi quá cân thức ăn trạm 2 [kiểm tra cân thức ăn]";
				AlarmList4[2,k1] := 'E30_2.Overload weightfood line 2 [check weightfood]';
			59: 
				AlarmList2[2,k1] := "E31_2.Lỗi quá cân sâu trạm 2 [kiểm tra cân sâu]";
				AlarmList4[2,k1] := 'E31_2.Overload weightlarvae line 2 [check weightlarvae]';
			61:
				AlarmList2[2,k1] := "E32_2.Lỗi ben hút/thả hũ đẩy ra trạm 2 [kiểm tra U1I7-12]";
				AlarmList4[2,k1] := 'E32_2.The cylinder sucking the jar is faulty line 2 [check U1I7-12]';
			62:
				AlarmList2[2,k1] := "E33_2.Lỗi Modbus thiết bị 1";
				AlarmList4[2,k1] := 'E33_2.Error Modbus device 1';
			63:
				AlarmList2[2,k1] := "E34_2.Lỗi Modbus thiết bị 2";
				AlarmList4[2,k1] := 'E34_2.Error Modbus device 2';
			64:
				AlarmList2[2,k1] := "E35_2.Lỗi Modbus thiết bị 3";
				AlarmList4[2,k1] := 'E35_2.Error Modbus device 3';
			67:
				AlarmList2[2,k1] := "E36_2.Lỗi Modbus thiết bị 6";
				AlarmList4[2,k1] := 'E36_2.Error Modbus device 6';
			71:
				AlarmList2[2,k1] := "E37_2.Lỗi đầu cân thức ăn Laumas";
				AlarmList4[2,k1] := 'E37_2.Error Laumas 1';
			72:
				AlarmList2[2,k1] := "E38_2.Lỗi đầu cân sâu Laumas";
				stErrorTxt3 := 'E38_2.Error Laumas 2';
			74:
				AlarmList2[2,k1] := "E39_2.Lỗi ben chặn sâu đẩy ra trạm 2 [kiểm tra U1I3-1]";
				AlarmList4[2,k1] := 'E39_2.The cylinder blocking worm extend  is faulty line 2';
			75:
				AlarmList2[2,k1] := "E40_2.Lỗi thiếu khí đầu vào [kiểm tra U1I7-13]";
				AlarmList4[2,k1] := 'E40_2.Error of lack of input air [check U1I7-13]';	
			78:
				AlarmList2[2,k1] := "E41_2.Lỗi hết thức ăn trạm 2";
				AlarmList4[2,k1] := 'E41_2.Error running out of food line 2';	
			79:
				AlarmList2[2,k1] := "E42_2.Lỗi hết sâu trạm 2";
				AlarmList4[2,k1] := 'E42_2.Error running out of larvae line 2';
			98:
				AlarmList2[2,k1] := "E98_2.Dừng khẩn [kiểm tra Emergency]"; 
				AlarmList4[2,k1] := 'E98_2.Emergency Stop [check Emergency]';
			99: 
				AlarmList2[2,k1] := "E99_2.Lỗi biến tần băng tải đầu ra [kiểm tra biến tần 3]";
				AlarmList4[2,k1] := 'E99_2.The inverter of conveyor ouy [check inverter 3]';
			108:
				AlarmList2[2,k1] := "W1_2.Cảnh báo hết hũ trạm 2 [kiểm tra U1I2-4]";
				AlarmList4[2,k1] := 'W1_2.Warning out of jar line 2 [check U1I2-4]';
			109:
				AlarmList2[2,k1] := "W2_2.Cảnh báo hết nắp trạm 2 [kiểm tra U1I3-2]";
				AlarmList4[2,k1] := 'W2_2.Warning out of lid line 2 [check U1I3-2]';
			110:
				AlarmList2[2,k1] := "W3_2.Cảnh báo hết thức ăn trạm 2";
				AlarmList4[2,k1] := 'W3_2.Warning running out of food line 2';
			111:
				AlarmList2[2,k1] := "W4_2.Cảnh báo cân quá khối lượng thức ăn trạm 2";
				AlarmList4[2,k1] := 'W4_2.Warning food weight exceeds limit line 2';
			112:
				AlarmList2[2,k1] := "W5_2.Cảnh báo hết sâu trạm 2";
				AlarmList4[2,k1] := 'W5_2.Warning running out of larvae line 2';
			113:
				AlarmList2[2,k1] := "W6_2.Canh bao can qua khoi luong sau tram 2";
				AlarmList4[2,k1] := 'W6_2.Warning larvae weight exceeds limit line 2';
			114:
				AlarmList2[2,k1] := "W7_2.Cảnh báo dập nắp không vô trạm 2 [kiểm tra U1I4-1]";
				AlarmList4[2,k1] := 'W7_2.Warning do not press lid inward line 2 [check U1I4-1]';
			115:
				AlarmList2[2,k1] := "W8_2.Cảnh báo mất kết nối với PC Advantech [kiểm tra PC]";
				AlarmList4[2,k1] := 'W8_2.Warning disconnect to PC Advantech [check PC]';	
		END_CASE
END_FOR
bWriteAlarm	:= FALSE;
END_IF
END_ACTION

ACTION steError_active:
PR_Line02.Stop();
bStatusStart2 := FALSE;
status := 'ERROR';
bfinish2 := TRUE;
IF a2 > 100 THEN
	a2 := 100;
END_IF
CASE nState2 OF 
	0:
		Reset_T(clk := bReset);
		IF Reset_T.Q THEN
			nState2 := 1;
		END_IF
	1:
		PR_Line02.Reset();
		timerReset(IN := TRUE, PT := T#500MS);
		IF nErrorIDList2[1].ErrorStatus = 1 THEN
			IF i <> 1 THEN
				FOR	k := a2 TO 2 BY -1 DO
				nErrorIDList2[k].nErrorID 	 := nErrorIDList2[k-1].nErrorID;
				nErrorIDList2[k].ErrorTime   := nErrorIDList2[k-1].ErrorTime;
				nErrorIDList2[k].ErrorStatus := nErrorIDList2[k-1].ErrorStatus;		
				END_FOR		
			END_IF 
			nState2 := 2;
		ELSE 
			nState2 := 3;
		END_IF
	2:
		bWriteAlarm	:= TRUE;
		PR_Line02.Reset();
		timerReset(IN := TRUE, PT := T#500MS);
		nErrorIDList2[1].nErrorID := nErrorID;
		nErrorIDList2[1].ErrorTime := SYSTEMTIME_TO_DT(GetLocalSystemTime.systemTime);
		nErrorIDList2[1].ErrorStatus := 0;
		a2 := a2  + 1;	
		nState2 := 3;
	3:
		PR_Line02.Reset();
		timerReset(IN := TRUE, PT := T#500MS);
		IF timerReset.Q THEN
			nState2 := 4;
		END_IF
	4:
		timerReset(IN := FALSE);
		Reset_T(clk := FALSE);
		traError := FALSE;
		nState2 := 0;
END_CASE

IF bReset THEN
	bError2 := FALSE;
	bWarning := FALSE;
	bSirens := FALSE;
	status := 'STOP';
	Error[1] := FALSE;
	Error[2] := FALSE;
	Error[6] := FALSE;
	Error[3] := FALSE;
END_IF

IF NOT bEmer THEN
	PR_Line02.Init();
END_IF

IF bTo_alarm_side2 AND NOT bTo_alarm_side THEN
	VisuElems.CURRENTVISU := 'N_Alarm_1';
	IF VisuElems.CURRENTVISU = 'N_Alarm_1' THEN
		bTo_alarm_side2 := FALSE;
	END_IF
END_IF
END_ACTION

ACTION steErrorCheck_active:

END_ACTION

ACTION steInit_active:
traInitDone := TRUE;
bStatusStart2 := FALSE;
END_ACTION

ACTION steModeAuto_active:
PR_Line02.Auto();
bResetmanual2 := TRUE;
IF bReset THEN
	bWarning2 := FALSE;
	bSirens	  := FALSE;
	bAlarm_Iot := FALSE;
	bWrn2	  := FALSE;
END_IF
END_ACTION

ACTION steModeManual_active:
PR_Line02.Manual();
PR_Line02.Check_reset();
END_ACTION

ACTION steModeSel_active:
IF VisuElems.CURRENTVISU = 'MAIN_LINE2' THEN
	bModeAuto := TRUE;
	bModeManual := FALSE;
END_IF

IF VisuElems.CURRENTVISU = 'N_FoodSupply2' OR VisuElems.CURRENTVISU = 'N_JarSupply2' OR VisuElems.CURRENTVISU = 'N_LidPressing2' OR
	VisuElems.CURRENTVISU = 'N_LidSupply2' OR VisuElems.CURRENTVISU = 'N_Tranfer2' OR VisuElems.CURRENTVISU = 'N_WormWeight2' THEN
	bModeAuto := FALSE;
	bModeManual := TRUE;
END_IF
PR_Line02.check();

IF bStart2 THEN
	bStart2 := FALSE;
END_IF
END_ACTION

END_PROGRAM

// ---- POUs/Recipe/PRG_MainRecipe1_1.TcPOU
PROGRAM PRG_MainRecipe1_1
VAR
	fbrecipe		: RecipeManCommands;
	NameSave		: STRING;
	NameLoad		: STRING;
	RecipeName		: STRING;
	RecipeNameIdx	: INT;
	r1				: INT;
	dLen			: INT;
	RecipeList 		: ARRAY[0..99] OF STRING;
	tTimer			: TON;
END_VAR

PRG_RecipeList1_1();

FOR r1 := 0 TO 99 DO
	dLen 			:= LEN(PRG_RecipeList1_1.filesList[r1].sFileName) - LEN('.Recipes_2.txtrecipe'); 
	RecipeList[r1] 	:= MID(PRG_RecipeList1_1.filesList[r1].sFileName,dLen,1);
END_FOR

IF bSave2 THEN
	fbRecipe.CreateRecipe('Recipes_2',NameSave);
	PRG_RecipeList1_1.bFirst	:= TRUE;
	bSave2 					:= FALSE;
ELSIF bLoad2 THEN
	RecipeName				:= RecipeList[RecipeNameIdx];
	fbRecipe.WriteRecipe('Recipes_2', RecipeName);
	PRG_RecipeList1_1.bFirst	:= TRUE;
	bLoad2 					:= FALSE;
ELSIF bDelete2 THEN
	RecipeName				:= RecipeList[RecipeNameIdx];
	fbRecipe.DeleteRecipe('Recipes_2', RecipeName);		
	PRG_RecipeList1_1.bFirst	:= TRUE;
	bDelete2 				:= FALSE;
END_IF

END_PROGRAM

// ---- POUs/Recipe/PRG_RecipeList1_1.TcPOU
PROGRAM PRG_RecipeList1_1
VAR_INPUT
		bFirst			: BOOL := TRUE;
END_VAR
VAR
	fbEnum				: FB_EnumFindFileList;
	filesList 			: ARRAY[0..99]  OF ST_FindFileEntry;
	bNext				: BOOL;
	bAbort				: BOOL;
	bBusy				: BOOL;
	bError				: BOOL;
	nErrID				: UDINT;
	bEOE				: BOOL;
	nFindFiles			: UDINT;
END_VAR

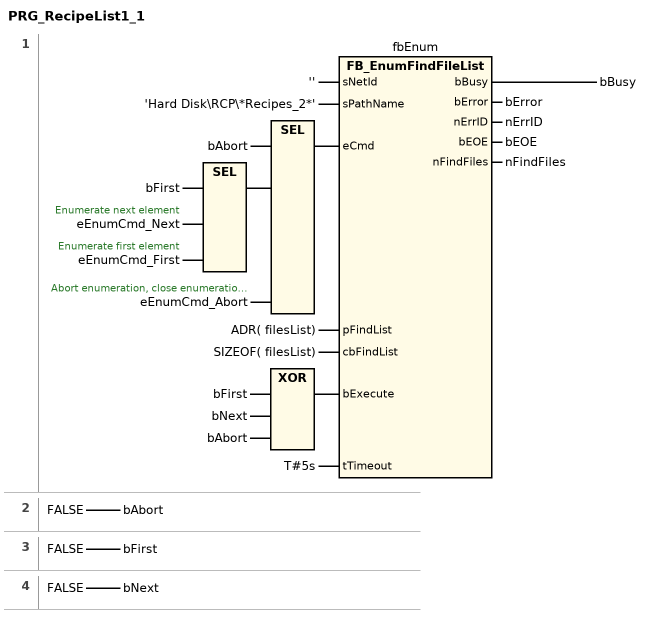
// NETWORK 1
//   eEnumCmd_Next: Enumerate next element
//   eEnumCmd_First: Enumerate first element
//   eEnumCmd_Abort: Abort enumeration, close enumeration handle.
fbEnum(
    sNetId := '',
    sPathName := 'Hard Disk\RCP\*Recipes_2*',
    eCmd := SEL(bAbort, SEL(bFirst, eEnumCmd_Next, eEnumCmd_First), eEnumCmd_Abort),
    pFindList := ADR( filesList),
    cbFindList := SIZEOF( filesList),
    bExecute := bFirst XOR bNext XOR bAbort,
    tTimeout := T#5s,
    bError => bError,
    nErrID => nErrID,
    bEOE => bEOE,
    nFindFiles => nFindFiles); // FB_EnumFindFileList
bBusy := fbEnum.bBusy;

// NETWORK 2
bAbort := FALSE;

// NETWORK 3
bFirst := FALSE;

// NETWORK 4
bNext := FALSE;

END_PROGRAM

// ---- POUs/Components/Sim Components/FB_Conveyor_Sim.TcPOU
FUNCTION_BLOCK FB_Conveyor_Sim IMPLEMENTS I_Conveyor
VAR_INPUT
END_VAR
VAR_OUTPUT
END_VAR
VAR
	bRunConveyor : BOOL;
	bIsRun		 : BOOL;
END_VAR

IF bRunConveyor THEN
	bIsRun := TRUE;
ELSE
	bIsRun := FALSE;
END_IF

PROPERTY IsRun : BOOL
GET
IsRun := bIsRun;
END_GET
END_PROPERTY

METHOD Start : BOOL
VAR_INPUT
END_VAR
bRunConveyor := TRUE;
END_METHOD

METHOD Stop : BOOL
VAR_INPUT
END_VAR
bRunConveyor := FALSE;
END_METHOD

END_FUNCTION_BLOCK

